RoboDK station: Sheet C - Top.rdk

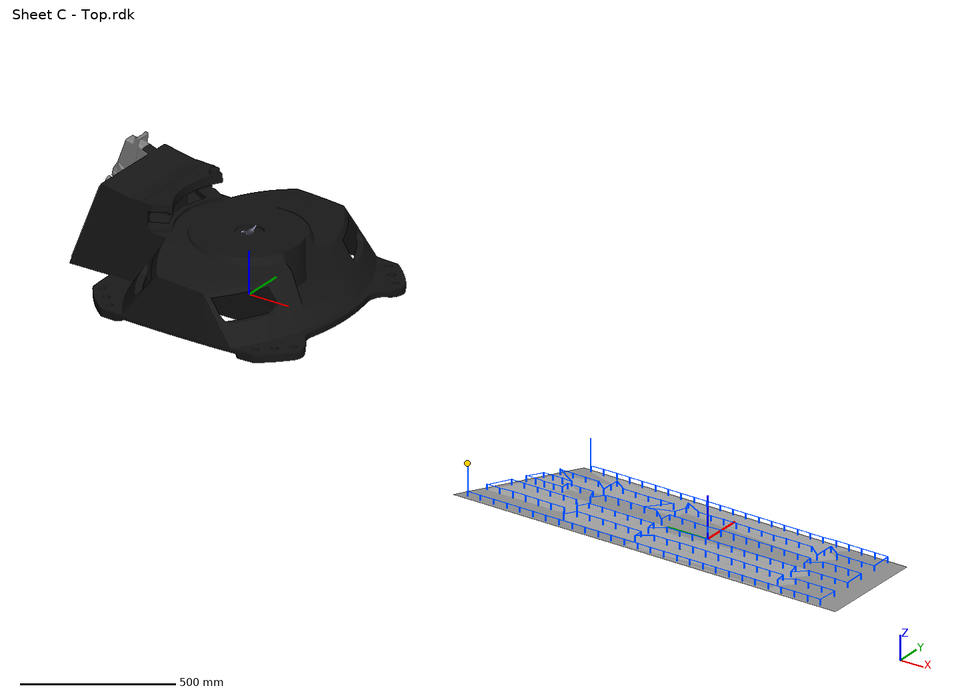
[picture v0: the station drawn from its stored meshes, robots at their saved joint values, targets as dots, program paths as lines]
Station Sheet C - Top (saved by RoboDK 5.2.3). Poses are relative to the parent item; angles as X-Y-Z fixed-axis rotations.
  - frame KUKA KR 210 R2700 extra Base at (0, 0, 0) mm
    - robot KUKA KR 210 R2700 extra: 6 axes, payload 210 kg, reach 2696 mm, repeatability 0.06 mm, weight 1068 kg
        joint limits [-185, -140, -120, -350, -125, -350] to [185, -5, 155, 350, 125, 350]; home [0, -90, 90, 0, 0, 0]; saved at [-11.417, -31.583, 137.817, -188.748, 54.991, -183.874]
      - tool Spindle, TCP at (32, 0, 260) mm, rotated rx 0 ry 39 rz 0 deg, size 157.3 x 72 x 259.9 mm
  - frame Frame 2 at (1800, 0, -372.68) mm, rotated rx 0 ry 0 rz 90 deg
    - object Box 1 - Sheet C -  Top at (0, 0, 0) mm, size 400 x 1500 x 0.8 mm, 1 curves, geometry from Box 1 - Sheet C -  Top.stl
    - object Sheet C-box 1 Hole positioning Top at (0, 0, 0) mm, 181 curves, geometry from Point 181
  - machining project Point settings: rotZ(0) | rotX(0)*rotY(0) | rotz(0)
  - program Point (916 instructions, listed below)
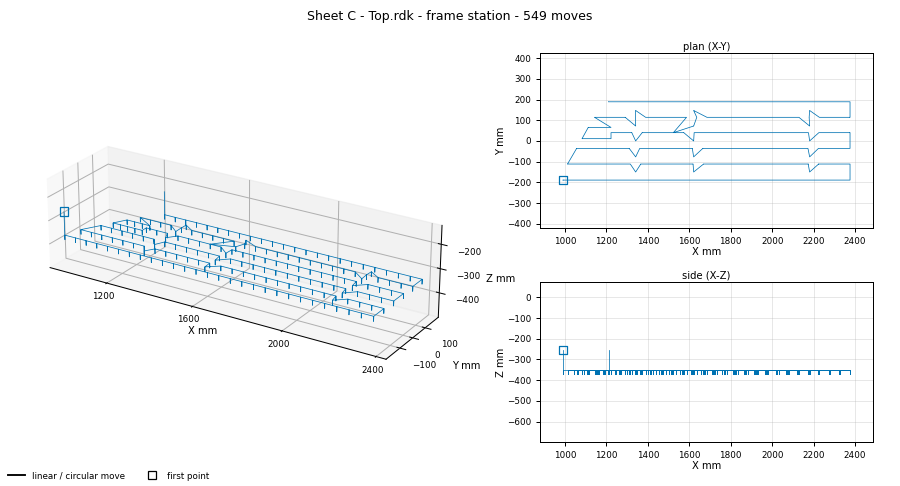
[picture p0: tool path of Sheet C - Top.rdk in frame station, 549 of 549 moves have a stored position in this frame; points joined in program order, loops and branches not executed]

--- program Point (robot KUKA KR 210 R2700 extra) ---
  Smooth(1)
  Set speed (1000.0 mm/s)
  Set Ref.: Frame 2
  Set Tool: Spindle
  Show Spindle
  MoveJ 1 to (-189, 810.01, 120) mm, rotated rx -180 ry 0 rz 90 deg; joints [14.788, -23.755, 145.264, -170.148, 69.845, -171.831]
  MoveL 2 to (-189, 810.01, 120) mm, rotated rx -180 ry 0 rz 90 deg; joints [14.788, -23.755, 145.264, -170.148, 69.845, -171.831]
  MoveL 3 to (-189, 810.01, 20) mm, rotated rx 180 ry 0 rz 90 deg; joints [14.788, -16.611, 140.997, -170.313, 72.681, -171.315]
  MoveL 4 to (-189, 810.01, 20) mm, rotated rx 180 ry 0 rz 90 deg; joints [14.788, -16.611, 140.997, -170.313, 72.681, -171.315]
  Set speed (50.0 mm/s)
  MoveL 5 to (-189, 810.01, 0) mm, rotated rx 180 ry 0 rz 90 deg; joints [14.788, -15.296, 140.112, -170.336, 73.105, -171.239]
  MoveL 6 to (-189, 810.01, 20) mm, rotated rx 180 ry 0 rz 90 deg; joints [14.788, -16.611, 140.997, -170.313, 72.681, -171.315]
  Set speed (1000.0 mm/s)
  MoveL 7 to (-189, 758.68, 20) mm, rotated rx 180 ry 0 rz 90 deg; joints [13.838, -18.904, 139.596, -170.729, 69.122, -172.492]
  Set speed (50.0 mm/s)
  MoveL 8 to (-189, 758.68, 0) mm, rotated rx -180 ry 0 rz 90 deg; joints [13.838, -17.57, 138.739, -170.758, 69.592, -172.41]
  MoveL 9 to (-189, 758.68, 20) mm, rotated rx 180 ry 0 rz 90 deg; joints [13.838, -18.904, 139.596, -170.729, 69.122, -172.492]
  Set speed (1000.0 mm/s)
  MoveL 10 to (-189, 707.34, 20) mm, rotated rx -180 ry 0 rz 90 deg; joints [13.001, -20.924, 138.071, -171.063, 65.686, -173.533]
  Set speed (50.0 mm/s)
  MoveL 11 to (-189, 707.34, 0) mm, rotated rx 180 ry 0 rz 90 deg; joints [13.001, -19.583, 137.241, -171.098, 66.19, -173.446]
  MoveL 12 to (-189, 707.34, 20) mm, rotated rx -180 ry 0 rz 90 deg; joints [13.001, -20.924, 138.071, -171.063, 65.686, -173.533]
  Set speed (1000.0 mm/s)
  MoveL 13 to (-189, 656.01, 20) mm, rotated rx 180 ry 0 rz 90 deg; joints [12.258, -22.682, 136.432, -171.327, 62.377, -174.462]
  Set speed (50.0 mm/s)
  MoveL 14 to (-189, 656.01, 0) mm, rotated rx 180 ry 0 rz 90 deg; joints [12.258, -21.344, 135.628, -171.369, 62.906, -174.371]
  MoveL 15 to (-189, 656.01, 20) mm, rotated rx 180 ry 0 rz 90 deg; joints [12.258, -22.682, 136.432, -171.327, 62.377, -174.462]
  Set speed (1000.0 mm/s)
  MoveL 16 to (-189, 604.68, 20) mm, rotated rx -180 ry 0 rz 90 deg; joints [11.594, -24.194, 134.688, -171.533, 59.195, -175.301]
  Set speed (50.0 mm/s)
  MoveL 17 to (-189, 604.68, 0) mm, rotated rx -180 ry 0 rz 90 deg; joints [11.594, -22.864, 133.91, -171.58, 59.74, -175.207]
  MoveL 18 to (-189, 604.68, 20) mm, rotated rx -180 ry 0 rz 90 deg; joints [11.594, -24.194, 134.688, -171.533, 59.195, -175.301]
  Set speed (1000.0 mm/s)
  MoveL 19 to (-189, 553.34, 20) mm, rotated rx -180 ry 0 rz 90 deg; joints [10.997, -25.475, 132.846, -171.687, 56.133, -176.067]
  Set speed (50.0 mm/s)
  MoveL 20 to (-189, 553.34, 0) mm, rotated rx 180 ry 0 rz 90 deg; joints [10.997, -24.16, 132.092, -171.741, 56.688, -175.97]
  MoveL 21 to (-189, 553.34, 20) mm, rotated rx -180 ry 0 rz 90 deg; joints [10.997, -25.475, 132.846, -171.687, 56.133, -176.067]
  Set speed (1000.0 mm/s)
  MoveL 22 to (-189, 502.01, 20) mm, rotated rx 180 ry 0 rz 90 deg; joints [10.458, -26.541, 130.913, -171.797, 53.186, -176.774]
  Set speed (50.0 mm/s)
  MoveL 23 to (-189, 502.01, 0) mm, rotated rx 180 ry 0 rz 90 deg; joints [10.458, -25.246, 130.183, -171.856, 53.746, -176.674]
  MoveL 24 to (-189, 502.01, 20) mm, rotated rx 180 ry 0 rz 90 deg; joints [10.458, -26.541, 130.913, -171.797, 53.186, -176.774]
  Set speed (1000.0 mm/s)
  MoveL 25 to (-189, 450.68, 20) mm, rotated rx -180 ry 0 rz 90 deg; joints [9.969, -27.41, 128.897, -171.865, 50.346, -177.434]
  Set speed (50.0 mm/s)
  MoveL 26 to (-189, 450.68, 0) mm, rotated rx 180 ry 0 rz 90 deg; joints [9.969, -26.137, 128.189, -171.931, 50.906, -177.33]
  MoveL 27 to (-189, 450.68, 20) mm, rotated rx -180 ry 0 rz 90 deg; joints [9.969, -27.41, 128.897, -171.865, 50.346, -177.434]
  Set speed (1000.0 mm/s)
  MoveL 28 to (-189, 399.34, 20) mm, rotated rx -180 ry 0 rz 90 deg; joints [9.523, -28.095, 126.8, -171.895, 47.604, -178.057]
  Set speed (50.0 mm/s)
  MoveL 29 to (-189, 399.34, 0) mm, rotated rx 180 ry 0 rz 90 deg; joints [9.523, -26.846, 126.113, -171.966, 48.16, -177.951]
  MoveL 30 to (-189, 399.34, 20) mm, rotated rx -180 ry 0 rz 90 deg; joints [9.523, -28.095, 126.8, -171.895, 47.604, -178.057]
  Set speed (1000.0 mm/s)
  MoveL 31 to (-189, 348.01, 20) mm, rotated rx 180 ry 0 rz 90 deg; joints [9.115, -28.611, 124.629, -171.887, 44.95, -178.653]
  Set speed (50.0 mm/s)
  MoveL 32 to (-189, 348.01, 0) mm, rotated rx 180 ry 0 rz 90 deg; joints [9.115, -27.388, 123.961, -171.965, 45.5, -178.543]
  MoveL 33 to (-189, 348.01, 20) mm, rotated rx 180 ry 0 rz 90 deg; joints [9.115, -28.611, 124.629, -171.887, 44.95, -178.653]
  Set speed (1000.0 mm/s)
  MoveL 34 to (-189, 296.68, 20) mm, rotated rx 180 ry 0 rz 90 deg; joints [8.741, -28.971, 122.385, -171.843, 42.377, -179.231]
  Set speed (50.0 mm/s)
  MoveL 35 to (-189, 296.68, 0) mm, rotated rx 180 ry 0 rz 90 deg; joints [8.741, -27.775, 121.736, -171.927, 42.919, -179.117]
  MoveL 36 to (-189, 296.68, 20) mm, rotated rx 180 ry 0 rz 90 deg; joints [8.741, -28.971, 122.385, -171.843, 42.377, -179.231]
  Set speed (1000.0 mm/s)
  MoveL 37 to (-189, 245.34, 20) mm, rotated rx 180 ry 0 rz 90 deg; joints [8.395, -29.188, 120.072, -171.76, 39.875, -179.799]
  Set speed (50.0 mm/s)
  MoveL 38 to (-189, 245.34, 0) mm, rotated rx 180 ry 0 rz 90 deg; joints [8.395, -28.018, 119.439, -171.851, 40.406, -179.68]
  MoveL 39 to (-189, 245.34, 20) mm, rotated rx 180 ry 0 rz 90 deg; joints [8.395, -29.188, 120.072, -171.76, 39.875, -179.799]
  Set speed (1000.0 mm/s)
  MoveL 40 to (-189, 194.01, 20) mm, rotated rx -180 ry 0 rz 90 deg; joints [8.076, -29.271, 117.69, -171.637, 37.436, -180.365]
  Set speed (50.0 mm/s)
  MoveL 41 to (-189, 194.01, 0) mm, rotated rx -180 ry 0 rz 90 deg; joints [8.076, -28.128, 117.073, -171.735, 37.956, -180.241]
  MoveL 42 to (-189, 194.01, 20) mm, rotated rx -180 ry 0 rz 90 deg; joints [8.076, -29.271, 117.69, -171.637, 37.436, -180.365]
  Set speed (1000.0 mm/s)
  MoveL 43 to (-189, 142.68, 20) mm, rotated rx -180 ry 0 rz 90 deg; joints [7.78, -29.229, 115.242, -171.469, 35.053, -180.939]
  Set speed (50.0 mm/s)
  MoveL 44 to (-189, 142.68, 0) mm, rotated rx 180 ry 0 rz 90 deg; joints [7.78, -28.112, 114.639, -171.576, 35.561, -180.808]
  MoveL 45 to (-189, 142.68, 20) mm, rotated rx -180 ry 0 rz 90 deg; joints [7.78, -29.229, 115.242, -171.469, 35.053, -180.939]
  Set speed (1000.0 mm/s)
  MoveL 46 to (-189, 91.34, 20) mm, rotated rx -180 ry 0 rz 90 deg; joints [7.505, -29.071, 112.726, -171.253, 32.718, -181.53]
  Set speed (50.0 mm/s)
  MoveL 47 to (-189, 91.34, 0) mm, rotated rx 180 ry 0 rz 90 deg; joints [7.505, -27.98, 112.135, -171.369, 33.212, -181.392]
  MoveL 48 to (-189, 91.34, 20) mm, rotated rx -180 ry 0 rz 90 deg; joints [7.505, -29.071, 112.726, -171.253, 32.718, -181.53]
  Set speed (1000.0 mm/s)
  MoveL 49 to (-189, 40.01, 20) mm, rotated rx -180 ry 0 rz 90 deg; joints [7.249, -28.804, 110.142, -170.978, 30.424, -182.151]
  Set speed (50.0 mm/s)
  MoveL 50 to (-189, 40.01, 0) mm, rotated rx -180 ry 0 rz 90 deg; joints [7.249, -27.738, 109.563, -171.106, 30.905, -182.002]
  MoveL 51 to (-189, 40.01, 20) mm, rotated rx -180 ry 0 rz 90 deg; joints [7.249, -28.804, 110.142, -170.978, 30.424, -182.151]
  Set speed (1000.0 mm/s)
  MoveL 52 to (-189, -11.32, 20) mm, rotated rx 180 ry 0 rz 90 deg; joints [7.009, -28.434, 107.49, -170.637, 28.165, -182.813]
  Set speed (50.0 mm/s)
  MoveL 53 to (-189, -11.32, 0) mm, rotated rx -180 ry 0 rz 90 deg; joints [7.009, -27.391, 106.92, -170.778, 28.632, -182.653]
  MoveL 54 to (-189, -11.32, 20) mm, rotated rx 180 ry 0 rz 90 deg; joints [7.009, -28.434, 107.49, -170.637, 28.165, -182.813]
  Set speed (1000.0 mm/s)
  MoveL 55 to (-189, -62.66, 20) mm, rotated rx 180 ry 0 rz 90 deg; joints [6.785, -27.964, 104.766, -170.212, 25.933, -183.536]
  Set speed (50.0 mm/s)
  MoveL 56 to (-189, -62.66, 0) mm, rotated rx 180 ry 0 rz 90 deg; joints [6.785, -26.945, 104.205, -170.369, 26.385, -183.361]
  MoveL 57 to (-189, -62.66, 20) mm, rotated rx 180 ry 0 rz 90 deg; joints [6.785, -27.964, 104.766, -170.212, 25.933, -183.536]
  Set speed (1000.0 mm/s)
  MoveL 58 to (-189, -113.99, 20) mm, rotated rx 180 ry 0 rz 90 deg; joints [6.574, -27.401, 101.968, -169.684, 23.725, -184.343]
  Set speed (50.0 mm/s)
  MoveL 59 to (-189, -113.99, 0) mm, rotated rx -180 ry 0 rz 90 deg; joints [6.574, -26.403, 101.414, -169.861, 24.162, -184.148]
  MoveL 60 to (-189, -113.99, 20) mm, rotated rx 180 ry 0 rz 90 deg; joints [6.574, -27.401, 101.968, -169.684, 23.725, -184.343]
  Set speed (1000.0 mm/s)
  MoveL 61 to (-189, -165.32, 20) mm, rotated rx -180 ry 0 rz 90 deg; joints [6.376, -26.745, 99.093, -169.022, 21.533, -185.265]
  Set speed (50.0 mm/s)
  MoveL 62 to (-189, -165.32, 0) mm, rotated rx -180 ry 0 rz 90 deg; joints [6.376, -25.768, 98.545, -169.226, 21.955, -185.046]
  MoveL 63 to (-189, -165.32, 20) mm, rotated rx -180 ry 0 rz 90 deg; joints [6.376, -26.745, 99.093, -169.022, 21.533, -185.265]
  Set speed (1000.0 mm/s)
  MoveL 64 to (-189, -216.66, 20) mm, rotated rx 180 ry 0 rz 90 deg; joints [6.19, -26, 96.135, -168.183, 19.352, -186.348]
  Set speed (50.0 mm/s)
  MoveL 65 to (-189, -216.66, 0) mm, rotated rx -180 ry 0 rz 90 deg; joints [6.19, -25.042, 95.592, -168.42, 19.758, -186.097]
  MoveL 66 to (-189, -216.66, 20) mm, rotated rx 180 ry 0 rz 90 deg; joints [6.19, -26, 96.135, -168.183, 19.352, -186.348]
  Set speed (1000.0 mm/s)
  MoveL 67 to (-189, -267.99, 20) mm, rotated rx 180 ry 0 rz 90 deg; joints [6.014, -25.166, 93.09, -167.099, 17.178, -187.662]
  Set speed (50.0 mm/s)
  MoveL 68 to (-189, -267.99, 0) mm, rotated rx 180 ry 0 rz 90 deg; joints [6.014, -24.226, 92.55, -167.382, 17.568, -187.366]
  MoveL 69 to (-189, -267.99, 20) mm, rotated rx 180 ry 0 rz 90 deg; joints [6.014, -25.166, 93.09, -167.099, 17.178, -187.662]
  Set speed (1000.0 mm/s)
  MoveL 70 to (-189, -319.32, 20) mm, rotated rx -180 ry 0 rz 90 deg; joints [5.848, -24.243, 89.949, -165.662, 15.007, -189.317]
  Set speed (50.0 mm/s)
  MoveL 71 to (-189, -319.32, 0) mm, rotated rx -180 ry 0 rz 90 deg; joints [5.848, -23.32, 89.411, -166.009, 15.38, -188.957]
  MoveL 72 to (-189, -319.32, 20) mm, rotated rx -180 ry 0 rz 90 deg; joints [5.848, -24.243, 89.949, -165.662, 15.007, -189.317]
  Set speed (1000.0 mm/s)
  MoveL 73 to (-189, -370.66, 20) mm, rotated rx 180 ry 0 rz 90 deg; joints [5.691, -23.23, 86.705, -163.687, 12.837, -191.497]
  Set speed (50.0 mm/s)
  MoveL 74 to (-189, -370.66, 0) mm, rotated rx 180 ry 0 rz 90 deg; joints [5.691, -22.323, 86.167, -164.131, 13.192, -191.043]
  MoveL 75 to (-189, -370.66, 20) mm, rotated rx 180 ry 0 rz 90 deg; joints [5.691, -23.23, 86.705, -163.687, 12.837, -191.497]
  Set speed (1000.0 mm/s)
  MoveL 76 to (-189, -421.99, 20) mm, rotated rx -180 ry 0 rz 90 deg; joints [5.542, -22.125, 83.347, -160.837, 10.67, -194.543]
  Set speed (50.0 mm/s)
  MoveL 77 to (-189, -421.99, 0) mm, rotated rx 180 ry 0 rz 90 deg; joints [5.542, -21.231, 82.807, -161.435, 11.004, -193.935]
  MoveL 78 to (-189, -421.99, 20) mm, rotated rx -180 ry 0 rz 90 deg; joints [5.542, -22.125, 83.347, -160.837, 10.67, -194.543]
  Set speed (1000.0 mm/s)
  MoveL 79 to (-189, -473.32, 20) mm, rotated rx 180 ry 0 rz 90 deg; joints [5.4, -20.924, 79.863, -156.425, 8.516, -199.141]
  Set speed (50.0 mm/s)
  MoveL 80 to (-189, -473.32, 0) mm, rotated rx -180 ry 0 rz 90 deg; joints [5.4, -20.042, 79.319, -157.295, 8.827, -198.261]
  MoveL 81 to (-189, -473.32, 20) mm, rotated rx 180 ry 0 rz 90 deg; joints [5.4, -20.924, 79.863, -156.425, 8.516, -199.141]
  Set speed (1000.0 mm/s)
  MoveL 82 to (-189, -524.66, 20) mm, rotated rx -180 ry 0 rz 90 deg; joints [5.266, -19.621, 76.236, -148.871, 6.415, -206.873]
  Set speed (50.0 mm/s)
  MoveL 83 to (-189, -524.66, 0) mm, rotated rx -180 ry 0 rz 90 deg; joints [5.266, -18.75, 75.686, -150.285, 6.691, -205.45]
  MoveL 84 to (-189, -524.66, 20) mm, rotated rx -180 ry 0 rz 90 deg; joints [5.266, -19.621, 76.236, -148.871, 6.415, -206.873]
  Set speed (1000.0 mm/s)
  MoveL 85 to (-189, -575.99, 20) mm, rotated rx -180 ry 0 rz 90 deg; joints [5.138, -18.208, 72.448, -134.025, 4.496, -221.889]
  Set speed (50.0 mm/s)
  MoveL 86 to (-189, -575.99, 0) mm, rotated rx 180 ry 0 rz 90 deg; joints [5.138, -17.345, 71.889, -136.67, 4.711, -219.236]
  MoveL 87 to (-189, -575.99, 20) mm, rotated rx -180 ry 0 rz 90 deg; joints [5.138, -18.208, 72.448, -134.025, 4.496, -221.889]
  Set speed (1000.0 mm/s)
  MoveL 88 to (-111.5, -575.99, 20) mm, rotated rx 180 ry 0 rz 90 deg; joints [3.036, -18.366, 72.866, -151.076, 3.952, -206.505]
  Set speed (50.0 mm/s)
  MoveL 89 to (-111.5, -575.99, 0) mm, rotated rx -180 ry 0 rz 90 deg; joints [3.036, -17.503, 72.308, -153.075, 4.222, -204.502]
  MoveL 90 to (-111.5, -575.99, 20) mm, rotated rx 180 ry 0 rz 90 deg; joints [3.036, -18.366, 72.866, -151.076, 3.952, -206.505]
  Set speed (1000.0 mm/s)
  MoveL 91 to (-111.5, -525.47, 20) mm, rotated rx 180 ry 0 rz 90 deg; joints [3.111, -19.749, 76.587, -161.307, 6.118, -196.175]
  Set speed (50.0 mm/s)
  MoveL 92 to (-111.5, -525.47, 0) mm, rotated rx 180 ry 0 rz 90 deg; joints [3.111, -18.877, 76.038, -162.225, 6.424, -195.252]
  MoveL 93 to (-111.5, -525.47, 20) mm, rotated rx 180 ry 0 rz 90 deg; joints [3.111, -19.749, 76.587, -161.307, 6.118, -196.175]
  Set speed (1000.0 mm/s)
  MoveL 94 to (-111.5, -474.95, 20) mm, rotated rx 180 ry 0 rz 90 deg; joints [3.19, -21.026, 80.154, -166.01, 8.328, -191.369]
  Set speed (50.0 mm/s)
  MoveL 95 to (-111.5, -474.95, 0) mm, rotated rx 180 ry 0 rz 90 deg; joints [3.19, -20.144, 79.61, -166.548, 8.657, -190.824]
  MoveL 96 to (-111.5, -474.95, 20) mm, rotated rx 180 ry 0 rz 90 deg; joints [3.19, -21.026, 80.154, -166.01, 8.328, -191.369]
  Set speed (1000.0 mm/s)
  MoveL 97 to (-111.5, -424.43, 20) mm, rotated rx -180 ry 0 rz 90 deg; joints [3.272, -22.205, 83.583, -168.669, 10.533, -188.601]
  Set speed (50.0 mm/s)
  MoveL 98 to (-111.5, -424.43, 0) mm, rotated rx -180 ry 0 rz 90 deg; joints [3.272, -21.31, 83.043, -169.032, 10.882, -188.232]
  MoveL 99 to (-111.5, -424.43, 20) mm, rotated rx -180 ry 0 rz 90 deg; joints [3.272, -22.205, 83.583, -168.669, 10.533, -188.601]
  Set speed (1000.0 mm/s)
  MoveL 100 to (-150, -380.99, 20) mm, rotated rx 180 ry 0 rz 90 deg; joints [4.498, -23.088, 86.263, -166.725, 12.41, -189.478]
  Set speed (50.0 mm/s)
  MoveL 101 to (-150, -380.99, 0) mm, rotated rx -180 ry 0 rz 90 deg; joints [4.498, -22.182, 85.725, -167.097, 12.768, -189.096]
  MoveL 102 to (-150, -380.99, 20) mm, rotated rx 180 ry 0 rz 90 deg; joints [4.498, -23.088, 86.263, -166.725, 12.41, -189.478]
  Set speed (1000.0 mm/s)
  MoveL 103 to (-111.5, -373.92, 20) mm, rotated rx -180 ry 0 rz 90 deg; joints [3.359, -23.29, 86.89, -170.365, 12.726, -186.791]
  Set speed (50.0 mm/s)
  MoveL 104 to (-111.5, -373.92, 0) mm, rotated rx 180 ry 0 rz 90 deg; joints [3.359, -22.381, 86.352, -170.632, 13.091, -186.518]
  MoveL 105 to (-111.5, -373.92, 20) mm, rotated rx -180 ry 0 rz 90 deg; joints [3.359, -23.29, 86.89, -170.365, 12.726, -186.791]
  Set speed (1000.0 mm/s)
  MoveL 106 to (-111.5, -323.4, 20) mm, rotated rx 180 ry 0 rz 90 deg; joints [3.45, -24.285, 90.088, -171.534, 14.907, -185.503]
  Set speed (50.0 mm/s)
  MoveL 107 to (-111.5, -323.4, 0) mm, rotated rx 180 ry 0 rz 90 deg; joints [3.45, -23.361, 89.549, -171.742, 15.288, -185.287]
  MoveL 108 to (-111.5, -323.4, 20) mm, rotated rx 180 ry 0 rz 90 deg; joints [3.45, -24.285, 90.088, -171.534, 14.907, -185.503]
  Set speed (1000.0 mm/s)
  MoveL 109 to (-111.5, -272.88, 20) mm, rotated rx 180 ry 0 rz 90 deg; joints [3.547, -25.193, 93.186, -172.383, 17.081, -184.527]
  Set speed (50.0 mm/s)
  MoveL 110 to (-111.5, -272.88, 0) mm, rotated rx 180 ry 0 rz 90 deg; joints [3.547, -24.253, 92.646, -172.552, 17.478, -184.35]
  MoveL 111 to (-111.5, -272.88, 20) mm, rotated rx 180 ry 0 rz 90 deg; joints [3.547, -25.193, 93.186, -172.383, 17.081, -184.527]
  Set speed (1000.0 mm/s)
  MoveL 112 to (-111.5, -222.36, 20) mm, rotated rx 180 ry 0 rz 90 deg; joints [3.649, -26.015, 96.192, -173.023, 19.252, -183.753]
  Set speed (50.0 mm/s)
  MoveL 113 to (-111.5, -222.36, 0) mm, rotated rx -180 ry 0 rz 90 deg; joints [3.649, -25.056, 95.649, -173.164, 19.664, -183.603]
  MoveL 114 to (-111.5, -222.36, 20) mm, rotated rx 180 ry 0 rz 90 deg; joints [3.649, -26.015, 96.192, -173.023, 19.252, -183.753]
  Set speed (1000.0 mm/s)
  MoveL 115 to (-111.5, -171.84, 20) mm, rotated rx 180 ry 0 rz 90 deg; joints [3.757, -26.75, 99.113, -173.518, 21.427, -183.116]
  Set speed (50.0 mm/s)
  MoveL 116 to (-111.5, -171.84, 0) mm, rotated rx 180 ry 0 rz 90 deg; joints [3.757, -25.772, 98.565, -173.639, 21.854, -182.985]
  MoveL 117 to (-111.5, -171.84, 20) mm, rotated rx 180 ry 0 rz 90 deg; joints [3.757, -26.75, 99.113, -173.518, 21.427, -183.116]
  Set speed (1000.0 mm/s)
  MoveL 118 to (-111.5, -121.32, 20) mm, rotated rx -180 ry 0 rz 90 deg; joints [3.872, -27.398, 101.954, -173.909, 23.611, -182.573]
  Set speed (50.0 mm/s)
  MoveL 119 to (-111.5, -121.32, 0) mm, rotated rx -180 ry 0 rz 90 deg; joints [3.872, -26.4, 101.401, -174.015, 24.053, -182.458]
  MoveL 120 to (-111.5, -121.32, 20) mm, rotated rx -180 ry 0 rz 90 deg; joints [3.872, -27.398, 101.954, -173.909, 23.611, -182.573]
  Set speed (1000.0 mm/s)
  MoveL 121 to (-111.5, -70.81, 20) mm, rotated rx 180 ry 0 rz 90 deg; joints [3.994, -27.956, 104.72, -174.221, 25.811, -182.099]
  Set speed (50.0 mm/s)
  MoveL 122 to (-111.5, -70.81, 0) mm, rotated rx 180 ry 0 rz 90 deg; joints [3.994, -26.937, 104.16, -174.315, 26.267, -181.995]
  MoveL 123 to (-111.5, -70.81, 20) mm, rotated rx 180 ry 0 rz 90 deg; joints [3.994, -27.956, 104.72, -174.221, 25.811, -182.099]
  Set speed (1000.0 mm/s)
  MoveL 124 to (-111.5, -20.29, 20) mm, rotated rx 180 ry 0 rz 90 deg; joints [4.125, -28.422, 107.415, -174.473, 28.031, -181.674]
  Set speed (50.0 mm/s)
  MoveL 125 to (-111.5, -20.29, 0) mm, rotated rx -180 ry 0 rz 90 deg; joints [4.125, -27.38, 106.846, -174.557, 28.502, -181.579]
  MoveL 126 to (-111.5, -20.29, 20) mm, rotated rx 180 ry 0 rz 90 deg; joints [4.125, -28.422, 107.415, -174.473, 28.031, -181.674]
  Set speed (1000.0 mm/s)
  MoveL 127 to (-111.5, 30.23, 20) mm, rotated rx -180 ry 0 rz 90 deg; joints [4.263, -28.792, 110.042, -174.676, 30.28, -181.285]
  Set speed (50.0 mm/s)
  MoveL 128 to (-111.5, 30.23, 0) mm, rotated rx -180 ry 0 rz 90 deg; joints [4.263, -27.726, 109.462, -174.752, 30.764, -181.197]
  MoveL 129 to (-111.5, 30.23, 20) mm, rotated rx -180 ry 0 rz 90 deg; joints [4.263, -28.792, 110.042, -174.676, 30.28, -181.285]
  Set speed (1000.0 mm/s)
  MoveL 130 to (-111.5, 80.75, 20) mm, rotated rx -180 ry 0 rz 90 deg; joints [4.412, -29.061, 112.601, -174.84, 32.563, -180.921]
  Set speed (50.0 mm/s)
  MoveL 131 to (-111.5, 80.75, 0) mm, rotated rx 180 ry 0 rz 90 deg; joints [4.412, -27.971, 112.011, -174.909, 33.06, -180.839]
  MoveL 132 to (-111.5, 80.75, 20) mm, rotated rx -180 ry 0 rz 90 deg; joints [4.412, -29.061, 112.601, -174.84, 32.563, -180.921]
  Set speed (1000.0 mm/s)
  MoveL 133 to (-111.5, 131.27, 20) mm, rotated rx -180 ry 0 rz 90 deg; joints [4.571, -29.223, 115.095, -174.97, 34.887, -180.575]
  Set speed (50.0 mm/s)
  MoveL 134 to (-111.5, 131.27, 0) mm, rotated rx -180 ry 0 rz 90 deg; joints [4.571, -28.108, 114.492, -175.033, 35.397, -180.497]
  MoveL 135 to (-111.5, 131.27, 20) mm, rotated rx -180 ry 0 rz 90 deg; joints [4.571, -29.223, 115.095, -174.97, 34.887, -180.575]
  Set speed (1000.0 mm/s)
  MoveL 136 to (-150, 179.01, 20) mm, rotated rx -180 ry 0 rz 90 deg; joints [6.355, -29.272, 117.215, -173.347, 36.956, -180.379]
  Set speed (50.0 mm/s)
  MoveL 137 to (-150, 179.01, 0) mm, rotated rx 180 ry 0 rz 90 deg; joints [6.355, -28.134, 116.6, -173.426, 37.476, -180.279]
  MoveL 138 to (-150, 179.01, 20) mm, rotated rx -180 ry 0 rz 90 deg; joints [6.355, -29.272, 117.215, -173.347, 36.956, -180.379]
  Set speed (1000.0 mm/s)
  MoveL 139 to (-111.5, 181.79, 20) mm, rotated rx 180 ry 0 rz 90 deg; joints [4.742, -29.272, 117.524, -175.07, 37.259, -180.239]
  Set speed (50.0 mm/s)
  MoveL 140 to (-111.5, 181.79, 0) mm, rotated rx -180 ry 0 rz 90 deg; joints [4.742, -28.13, 116.908, -175.129, 37.782, -180.165]
  MoveL 141 to (-111.5, 181.79, 20) mm, rotated rx 180 ry 0 rz 90 deg; joints [4.742, -29.272, 117.524, -175.07, 37.259, -180.239]
  Set speed (1000.0 mm/s)
  MoveL 142 to (-111.5, 232.31, 20) mm, rotated rx -180 ry 0 rz 90 deg; joints [4.926, -29.199, 119.889, -175.145, 39.687, -179.907]
  Set speed (50.0 mm/s)
  MoveL 143 to (-111.5, 232.31, 0) mm, rotated rx 180 ry 0 rz 90 deg; joints [4.926, -28.031, 119.257, -175.199, 40.222, -179.837]
  MoveL 144 to (-111.5, 232.31, 20) mm, rotated rx -180 ry 0 rz 90 deg; joints [4.926, -29.199, 119.889, -175.145, 39.687, -179.907]
  Set speed (1000.0 mm/s)
  MoveL 145 to (-111.5, 282.82, 20) mm, rotated rx 180 ry 0 rz 90 deg; joints [5.125, -28.996, 122.187, -175.197, 42.179, -179.576]
  Set speed (50.0 mm/s)
  MoveL 146 to (-111.5, 282.82, 0) mm, rotated rx 180 ry 0 rz 90 deg; joints [5.125, -27.802, 121.539, -175.247, 42.724, -179.508]
  MoveL 147 to (-111.5, 282.82, 20) mm, rotated rx 180 ry 0 rz 90 deg; joints [5.125, -28.996, 122.187, -175.197, 42.179, -179.576]
  Set speed (1000.0 mm/s)
  MoveL 148 to (-111.5, 333.34, 20) mm, rotated rx -180 ry 0 rz 90 deg; joints [5.341, -28.652, 124.419, -175.226, 44.745, -179.239]
  Set speed (50.0 mm/s)
  MoveL 149 to (-111.5, 333.34, 0) mm, rotated rx 180 ry 0 rz 90 deg; joints [5.341, -27.431, 123.754, -175.272, 45.298, -179.174]
  MoveL 150 to (-111.5, 333.34, 20) mm, rotated rx -180 ry 0 rz 90 deg; joints [5.341, -28.652, 124.419, -175.226, 44.745, -179.239]
  Set speed (1000.0 mm/s)
  MoveL 151 to (-111.5, 383.86, 20) mm, rotated rx -180 ry 0 rz 90 deg; joints [5.576, -28.155, 126.582, -175.234, 47.393, -178.891]
  Set speed (50.0 mm/s)
  MoveL 152 to (-111.5, 383.86, 0) mm, rotated rx 180 ry 0 rz 90 deg; joints [5.576, -26.909, 125.897, -175.277, 47.952, -178.829]
  MoveL 153 to (-111.5, 383.86, 20) mm, rotated rx -180 ry 0 rz 90 deg; joints [5.576, -28.155, 126.582, -175.234, 47.393, -178.891]
  Set speed (1000.0 mm/s)
  MoveL 154 to (-111.5, 434.38, 20) mm, rotated rx -180 ry 0 rz 90 deg; joints [5.832, -27.493, 128.672, -175.221, 50.133, -178.529]
  Set speed (50.0 mm/s)
  MoveL 155 to (-111.5, 434.38, 0) mm, rotated rx 180 ry 0 rz 90 deg; joints [5.832, -26.222, 127.967, -175.259, 50.696, -178.468]
  MoveL 156 to (-111.5, 434.38, 20) mm, rotated rx -180 ry 0 rz 90 deg; joints [5.832, -27.493, 128.672, -175.221, 50.133, -178.529]
  Set speed (1000.0 mm/s)
  MoveL 157 to (-150, 459.01, 20) mm, rotated rx 180 ry 0 rz 90 deg; joints [8.003, -27.183, 129.476, -173.545, 51.198, -177.82]
  Set speed (50.0 mm/s)
  MoveL 158 to (-150, 459.01, 0) mm, rotated rx -180 ry 0 rz 90 deg; joints [8.003, -25.903, 128.762, -173.595, 51.76, -177.739]
  MoveL 159 to (-150, 459.01, 20) mm, rotated rx 180 ry 0 rz 90 deg; joints [8.003, -27.183, 129.476, -173.545, 51.198, -177.82]
  Set speed (1000.0 mm/s)
  MoveL 160 to (-111.5, 484.9, 20) mm, rotated rx 180 ry 0 rz 90 deg; joints [6.113, -26.65, 130.687, -175.185, 52.975, -178.146]
  Set speed (50.0 mm/s)
  MoveL 161 to (-111.5, 484.9, 0) mm, rotated rx 180 ry 0 rz 90 deg; joints [6.113, -25.357, 129.96, -175.22, 53.538, -178.087]
  MoveL 162 to (-111.5, 484.9, 20) mm, rotated rx 180 ry 0 rz 90 deg; joints [6.113, -26.65, 130.687, -175.185, 52.975, -178.146]
  Set speed (1000.0 mm/s)
  MoveL 163 to (-111.5, 535.42, 20) mm, rotated rx -180 ry 0 rz 90 deg; joints [6.423, -25.612, 132.621, -175.125, 55.929, -177.736]
  Set speed (50.0 mm/s)
  MoveL 164 to (-111.5, 535.42, 0) mm, rotated rx 180 ry 0 rz 90 deg; joints [6.423, -24.3, 131.87, -175.157, 56.488, -177.679]
  MoveL 165 to (-111.5, 535.42, 20) mm, rotated rx -180 ry 0 rz 90 deg; joints [6.423, -25.612, 132.621, -175.125, 55.929, -177.736]
  Set speed (1000.0 mm/s)
  MoveL 166 to (-111.5, 585.94, 20) mm, rotated rx -180 ry 0 rz 90 deg; joints [6.765, -24.362, 134.468, -175.039, 59.005, -177.293]
  Set speed (50.0 mm/s)
  MoveL 167 to (-111.5, 585.94, 0) mm, rotated rx 180 ry 0 rz 90 deg; joints [6.765, -23.034, 133.693, -175.067, 59.556, -177.237]
  MoveL 168 to (-111.5, 585.94, 20) mm, rotated rx -180 ry 0 rz 90 deg; joints [6.765, -24.362, 134.468, -175.039, 59.005, -177.293]
  Set speed (1000.0 mm/s)
  MoveL 169 to (-111.5, 636.45, 20) mm, rotated rx 180 ry 0 rz 90 deg; joints [7.145, -22.883, 136.221, -174.924, 62.213, -176.807]
  Set speed (50.0 mm/s)
  MoveL 170 to (-111.5, 636.45, 0) mm, rotated rx 180 ry 0 rz 90 deg; joints [7.145, -21.545, 135.421, -174.949, 62.748, -176.754]
  MoveL 171 to (-111.5, 636.45, 20) mm, rotated rx 180 ry 0 rz 90 deg; joints [7.145, -22.883, 136.221, -174.924, 62.213, -176.807]
  Set speed (1000.0 mm/s)
  MoveL 172 to (-111.5, 686.97, 20) mm, rotated rx 180 ry 0 rz 90 deg; joints [7.57, -21.156, 137.874, -174.775, 65.563, -176.27]
  Set speed (50.0 mm/s)
  MoveL 173 to (-111.5, 686.97, 0) mm, rotated rx 180 ry 0 rz 90 deg; joints [7.57, -19.815, 137.047, -174.796, 66.074, -176.219]
  MoveL 174 to (-111.5, 686.97, 20) mm, rotated rx 180 ry 0 rz 90 deg; joints [7.57, -21.156, 137.874, -174.775, 65.563, -176.27]
  Set speed (1000.0 mm/s)
  MoveL 175 to (-111.5, 737.49, 20) mm, rotated rx -180 ry 0 rz 90 deg; joints [8.049, -19.165, 139.416, -174.586, 69.06, -175.668]
  Set speed (50.0 mm/s)
  MoveL 176 to (-111.5, 737.49, 0) mm, rotated rx -180 ry 0 rz 90 deg; joints [8.049, -17.831, 138.562, -174.603, 69.538, -175.62]
  MoveL 177 to (-111.5, 737.49, 20) mm, rotated rx -180 ry 0 rz 90 deg; joints [8.049, -19.165, 139.416, -174.586, 69.06, -175.668]
  Set speed (1000.0 mm/s)
  MoveL 178 to (-111.5, 788.01, 20) mm, rotated rx 180 ry 0 rz 90 deg; joints [8.592, -16.895, 140.838, -174.349, 72.706, -174.988]
  Set speed (50.0 mm/s)
  MoveL 179 to (-111.5, 788.01, 0) mm, rotated rx 180 ry 0 rz 90 deg; joints [8.592, -15.578, 139.957, -174.362, 73.141, -174.943]
  MoveL 180 to (-111.5, 788.01, 20) mm, rotated rx 180 ry 0 rz 90 deg; joints [8.592, -16.895, 140.838, -174.349, 72.706, -174.988]
  Set speed (1000.0 mm/s)
  MoveL 181 to (-36, 744.01, 20) mm, rotated rx -180 ry 0 rz 90 deg; joints [2.636, -18.579, 139.814, -178.237, 70.214, -178.548]
  Set speed (50.0 mm/s)
  MoveL 182 to (-36, 744.01, 0) mm, rotated rx 180 ry 0 rz 90 deg; joints [2.636, -17.248, 138.952, -178.242, 70.683, -178.532]
  MoveL 183 to (-36, 744.01, 20) mm, rotated rx -180 ry 0 rz 90 deg; joints [2.636, -18.579, 139.814, -178.237, 70.214, -178.548]
  Set speed (1000.0 mm/s)
  MoveL 184 to (-36, 693.24, 20) mm, rotated rx 180 ry 0 rz 90 deg; joints [2.476, -20.67, 138.281, -178.303, 66.594, -178.75]
  Set speed (50.0 mm/s)
  MoveL 185 to (-36, 693.24, 0) mm, rotated rx -180 ry 0 rz 90 deg; joints [2.476, -19.33, 137.447, -178.309, 67.1, -178.734]
  MoveL 186 to (-36, 693.24, 20) mm, rotated rx 180 ry 0 rz 90 deg; joints [2.476, -20.67, 138.281, -178.303, 66.594, -178.75]
  Set speed (1000.0 mm/s)
  MoveL 187 to (-36, 642.47, 20) mm, rotated rx 180 ry 0 rz 90 deg; joints [2.333, -22.484, 136.635, -178.354, 63.137, -178.93]
  Set speed (50.0 mm/s)
  MoveL 188 to (-36, 642.47, 0) mm, rotated rx -180 ry 0 rz 90 deg; joints [2.333, -21.145, 135.828, -178.362, 63.669, -178.913]
  MoveL 189 to (-36, 642.47, 20) mm, rotated rx 180 ry 0 rz 90 deg; joints [2.333, -22.484, 136.635, -178.354, 63.137, -178.93]
  Set speed (1000.0 mm/s)
  MoveL 190 to (-36, 591.7, 20) mm, rotated rx -180 ry 0 rz 90 deg; joints [2.207, -24.039, 134.884, -178.394, 59.834, -179.092]
  Set speed (50.0 mm/s)
  MoveL 191 to (-36, 591.7, 0) mm, rotated rx 180 ry 0 rz 90 deg; joints [2.207, -22.709, 134.103, -178.403, 60.383, -179.074]
  MoveL 192 to (-36, 591.7, 20) mm, rotated rx -180 ry 0 rz 90 deg; joints [2.207, -24.039, 134.884, -178.394, 59.834, -179.092]
  Set speed (1000.0 mm/s)
  MoveL 193 to (-36, 540.93, 20) mm, rotated rx -180 ry 0 rz 90 deg; joints [2.093, -25.355, 133.037, -178.424, 56.674, -179.239]
  Set speed (50.0 mm/s)
  MoveL 194 to (-36, 540.93, 0) mm, rotated rx -180 ry 0 rz 90 deg; joints [2.093, -24.038, 132.281, -178.434, 57.234, -179.221]
  MoveL 195 to (-36, 540.93, 20) mm, rotated rx -180 ry 0 rz 90 deg; joints [2.093, -25.355, 133.037, -178.424, 56.674, -179.239]
  Set speed (1000.0 mm/s)
  MoveL 196 to (-36, 490.16, 20) mm, rotated rx 180 ry 0 rz 90 deg; joints [1.991, -26.448, 131.102, -178.445, 53.646, -179.375]
  Set speed (50.0 mm/s)
  MoveL 197 to (-36, 490.16, 0) mm, rotated rx 180 ry 0 rz 90 deg; joints [1.991, -25.151, 130.37, -178.456, 54.211, -179.356]
  MoveL 198 to (-36, 490.16, 20) mm, rotated rx 180 ry 0 rz 90 deg; joints [1.991, -26.448, 131.102, -178.445, 53.646, -179.375]
  Set speed (1000.0 mm/s)
  MoveL 199 to (-77, 459.01, 20) mm, rotated rx -180 ry 0 rz 90 deg; joints [4.128, -27.054, 129.786, -176.691, 51.705, -178.842]
  Set speed (50.0 mm/s)
  MoveL 200 to (-77, 459.01, 0) mm, rotated rx -180 ry 0 rz 90 deg; joints [4.128, -25.771, 129.069, -176.717, 52.27, -178.801]
  MoveL 201 to (-77, 459.01, 20) mm, rotated rx -180 ry 0 rz 90 deg; joints [4.128, -27.054, 129.786, -176.691, 51.705, -178.842]
  Set speed (1000.0 mm/s)
  MoveL 202 to (-36, 439.39, 20) mm, rotated rx -180 ry 0 rz 90 deg; joints [1.898, -27.338, 129.083, -178.458, 50.74, -179.501]
  Set speed (50.0 mm/s)
  MoveL 203 to (-36, 439.39, 0) mm, rotated rx 180 ry 0 rz 90 deg; joints [1.898, -26.063, 128.374, -178.47, 51.305, -179.482]
  MoveL 204 to (-36, 439.39, 20) mm, rotated rx -180 ry 0 rz 90 deg; joints [1.898, -27.338, 129.083, -178.458, 50.74, -179.501]
  Set speed (1000.0 mm/s)
  MoveL 205 to (-36, 388.63, 20) mm, rotated rx 180 ry 0 rz 90 deg; joints [1.813, -28.041, 126.988, -178.463, 47.943, -179.62]
  Set speed (50.0 mm/s)
  MoveL 206 to (-36, 388.63, 0) mm, rotated rx -180 ry 0 rz 90 deg; joints [1.813, -26.791, 126.299, -178.477, 48.505, -179.6]
  MoveL 207 to (-36, 388.63, 20) mm, rotated rx 180 ry 0 rz 90 deg; joints [1.813, -28.041, 126.988, -178.463, 47.943, -179.62]
  Set speed (1000.0 mm/s)
  MoveL 208 to (-36, 337.86, 20) mm, rotated rx 180 ry 0 rz 90 deg; joints [1.736, -28.573, 124.819, -178.462, 45.244, -179.734]
  Set speed (50.0 mm/s)
  MoveL 209 to (-36, 337.86, 0) mm, rotated rx 180 ry 0 rz 90 deg; joints [1.736, -27.348, 124.15, -178.477, 45.8, -179.713]
  MoveL 210 to (-36, 337.86, 20) mm, rotated rx 180 ry 0 rz 90 deg; joints [1.736, -28.573, 124.819, -178.462, 45.244, -179.734]
  Set speed (1000.0 mm/s)
  MoveL 211 to (-36, 287.09, 20) mm, rotated rx 180 ry 0 rz 90 deg; joints [1.664, -28.946, 122.58, -178.453, 42.632, -179.844]
  Set speed (50.0 mm/s)
  MoveL 212 to (-36, 287.09, 0) mm, rotated rx 180 ry 0 rz 90 deg; joints [1.664, -27.748, 121.929, -178.469, 43.179, -179.823]
  MoveL 213 to (-36, 287.09, 20) mm, rotated rx 180 ry 0 rz 90 deg; joints [1.664, -28.946, 122.58, -178.453, 42.632, -179.844]
  Set speed (1000.0 mm/s)
  MoveL 214 to (-36, 236.32, 20) mm, rotated rx -180 ry 0 rz 90 deg; joints [1.599, -29.175, 120.273, -178.438, 40.097, -179.952]
  Set speed (50.0 mm/s)
  MoveL 215 to (-36, 236.32, 0) mm, rotated rx 180 ry 0 rz 90 deg; joints [1.599, -28.003, 119.639, -178.455, 40.635, -179.93]
  MoveL 216 to (-36, 236.32, 20) mm, rotated rx -180 ry 0 rz 90 deg; joints [1.599, -29.175, 120.273, -178.438, 40.097, -179.952]
  Set speed (1000.0 mm/s)
  MoveL 217 to (-36, 185.55, 20) mm, rotated rx -180 ry 0 rz 90 deg; joints [1.538, -29.268, 117.899, -178.414, 37.631, -180.06]
  Set speed (50.0 mm/s)
  MoveL 218 to (-36, 185.55, 0) mm, rotated rx -180 ry 0 rz 90 deg; joints [1.538, -28.123, 117.281, -178.433, 38.158, -180.037]
  MoveL 219 to (-36, 185.55, 20) mm, rotated rx -180 ry 0 rz 90 deg; joints [1.538, -29.268, 117.899, -178.414, 37.631, -180.06]
  Set speed (1000.0 mm/s)
  MoveL 220 to (-77, 179.01, 20) mm, rotated rx -180 ry 0 rz 90 deg; joints [3.272, -29.272, 117.507, -176.597, 37.238, -180.166]
  Set speed (50.0 mm/s)
  MoveL 221 to (-77, 179.01, 0) mm, rotated rx 180 ry 0 rz 90 deg; joints [3.272, -28.131, 116.891, -176.638, 37.762, -180.116]
  MoveL 222 to (-77, 179.01, 20) mm, rotated rx -180 ry 0 rz 90 deg; joints [3.272, -29.272, 117.507, -176.597, 37.238, -180.166]
  Set speed (1000.0 mm/s)
  MoveL 223 to (-36, 134.78, 20) mm, rotated rx 180 ry 0 rz 90 deg; joints [1.482, -29.238, 115.461, -178.383, 35.225, -180.169]
  Set speed (50.0 mm/s)
  MoveL 224 to (-36, 134.78, 0) mm, rotated rx -180 ry 0 rz 90 deg; joints [1.482, -28.118, 114.856, -178.403, 35.739, -180.144]
  MoveL 225 to (-36, 134.78, 20) mm, rotated rx 180 ry 0 rz 90 deg; joints [1.482, -29.238, 115.461, -178.383, 35.225, -180.169]
  Set speed (1000.0 mm/s)
  MoveL 226 to (-36, 84.01, 20) mm, rotated rx -180 ry 0 rz 90 deg; joints [1.43, -29.09, 112.957, -178.342, 32.869, -180.282]
  Set speed (50.0 mm/s)
  MoveL 227 to (-36, 84.01, 0) mm, rotated rx 180 ry 0 rz 90 deg; joints [1.43, -27.997, 112.365, -178.364, 33.37, -180.255]
  MoveL 228 to (-36, 84.01, 20) mm, rotated rx -180 ry 0 rz 90 deg; joints [1.43, -29.09, 112.957, -178.342, 32.869, -180.282]
  Set speed (1000.0 mm/s)
  MoveL 229 to (-36, 33.24, 20) mm, rotated rx 180 ry 0 rz 90 deg; joints [1.382, -28.834, 110.387, -178.29, 30.557, -180.399]
  Set speed (50.0 mm/s)
  MoveL 230 to (-36, 33.24, 0) mm, rotated rx 180 ry 0 rz 90 deg; joints [1.382, -27.765, 109.807, -178.314, 31.044, -180.371]
  MoveL 231 to (-36, 33.24, 20) mm, rotated rx 180 ry 0 rz 90 deg; joints [1.382, -28.834, 110.387, -178.29, 30.557, -180.399]
  Set speed (1000.0 mm/s)
  MoveL 232 to (-36, -17.53, 20) mm, rotated rx -180 ry 0 rz 90 deg; joints [1.336, -28.474, 107.75, -178.225, 28.28, -180.525]
  Set speed (50.0 mm/s)
  MoveL 233 to (-36, -17.53, 0) mm, rotated rx -180 ry 0 rz 90 deg; joints [1.336, -27.429, 107.18, -178.252, 28.754, -180.494]
  MoveL 234 to (-36, -17.53, 20) mm, rotated rx -180 ry 0 rz 90 deg; joints [1.336, -28.474, 107.75, -178.225, 28.28, -180.525]
  Set speed (1000.0 mm/s)
  MoveL 235 to (-36, -68.3, 20) mm, rotated rx -180 ry 0 rz 90 deg; joints [1.294, -28.016, 105.045, -178.145, 26.033, -180.662]
  Set speed (50.0 mm/s)
  MoveL 236 to (-36, -68.3, 0) mm, rotated rx -180 ry 0 rz 90 deg; joints [1.294, -26.994, 104.483, -178.175, 26.493, -180.628]
  MoveL 237 to (-36, -68.3, 20) mm, rotated rx -180 ry 0 rz 90 deg; joints [1.294, -28.016, 105.045, -178.145, 26.033, -180.662]
  Set speed (1000.0 mm/s)
  MoveL 238 to (-36, -119.07, 20) mm, rotated rx -180 ry 0 rz 90 deg; joints [1.254, -27.465, 102.267, -178.045, 23.808, -180.814]
  Set speed (50.0 mm/s)
  MoveL 239 to (-36, -119.07, 0) mm, rotated rx 180 ry 0 rz 90 deg; joints [1.254, -26.464, 101.712, -178.079, 24.253, -180.777]
  MoveL 240 to (-36, -119.07, 20) mm, rotated rx -180 ry 0 rz 90 deg; joints [1.254, -27.465, 102.267, -178.045, 23.808, -180.814]
  Set speed (1000.0 mm/s)
  MoveL 241 to (-36, -169.84, 20) mm, rotated rx 180 ry 0 rz 90 deg; joints [1.216, -26.822, 99.414, -177.92, 21.598, -180.988]
  Set speed (50.0 mm/s)
  MoveL 242 to (-36, -169.84, 0) mm, rotated rx 180 ry 0 rz 90 deg; joints [1.216, -25.842, 98.866, -177.959, 22.03, -180.947]
  MoveL 243 to (-36, -169.84, 20) mm, rotated rx 180 ry 0 rz 90 deg; joints [1.216, -26.822, 99.414, -177.92, 21.598, -180.988]
  Set speed (1000.0 mm/s)
  MoveL 244 to (-36, -220.61, 20) mm, rotated rx 180 ry 0 rz 90 deg; joints [1.181, -26.091, 96.481, -177.762, 19.398, -181.193]
  Set speed (50.0 mm/s)
  MoveL 245 to (-36, -220.61, 0) mm, rotated rx -180 ry 0 rz 90 deg; joints [1.181, -25.13, 95.938, -177.807, 19.815, -181.145]
  MoveL 246 to (-36, -220.61, 20) mm, rotated rx 180 ry 0 rz 90 deg; joints [1.181, -26.091, 96.481, -177.762, 19.398, -181.193]
  Set speed (1000.0 mm/s)
  MoveL 247 to (-36, -271.37, 20) mm, rotated rx -180 ry 0 rz 90 deg; joints [1.147, -25.272, 93.464, -177.558, 17.201, -181.442]
  Set speed (50.0 mm/s)
  MoveL 248 to (-36, -271.37, 0) mm, rotated rx -180 ry 0 rz 90 deg; joints [1.147, -24.33, 92.923, -177.612, 17.602, -181.385]
  MoveL 249 to (-36, -271.37, 20) mm, rotated rx -180 ry 0 rz 90 deg; joints [1.147, -25.272, 93.464, -177.558, 17.201, -181.442]
  Set speed (1000.0 mm/s)
  MoveL 250 to (-36, -322.14, 20) mm, rotated rx 180 ry 0 rz 90 deg; joints [1.116, -24.365, 90.354, -177.285, 14.999, -181.755]
  Set speed (50.0 mm/s)
  MoveL 251 to (-36, -322.14, 0) mm, rotated rx -180 ry 0 rz 90 deg; joints [1.116, -23.44, 89.815, -177.352, 15.385, -181.686]
  MoveL 252 to (-36, -322.14, 20) mm, rotated rx 180 ry 0 rz 90 deg; joints [1.116, -24.365, 90.354, -177.285, 14.999, -181.755]
  Set speed (1000.0 mm/s)
  MoveL 253 to (-36, -372.91, 20) mm, rotated rx -180 ry 0 rz 90 deg; joints [1.086, -23.371, 87.143, -176.91, 12.786, -182.169]
  Set speed (50.0 mm/s)
  MoveL 254 to (-36, -372.91, 0) mm, rotated rx -180 ry 0 rz 90 deg; joints [1.086, -22.461, 86.605, -176.996, 13.157, -182.081]
  MoveL 255 to (-36, -372.91, 20) mm, rotated rx -180 ry 0 rz 90 deg; joints [1.086, -23.371, 87.143, -176.91, 12.786, -182.169]
  Set speed (1000.0 mm/s)
  MoveL 256 to (-77, -380.99, 20) mm, rotated rx 180 ry 0 rz 90 deg; joints [2.312, -23.179, 86.544, -173.224, 12.427, -184.822]
  Set speed (50.0 mm/s)
  MoveL 257 to (-77, -380.99, 0) mm, rotated rx 180 ry 0 rz 90 deg; joints [2.312, -22.272, 86.006, -173.416, 12.793, -184.625]
  MoveL 258 to (-77, -380.99, 20) mm, rotated rx 180 ry 0 rz 90 deg; joints [2.312, -23.179, 86.544, -173.224, 12.427, -184.822]
  Set speed (1000.0 mm/s)
  MoveL 259 to (-36, -423.68, 20) mm, rotated rx -180 ry 0 rz 90 deg; joints [1.058, -22.285, 83.823, -176.363, 10.554, -182.753]
  Set speed (50.0 mm/s)
  MoveL 260 to (-36, -423.68, 0) mm, rotated rx 180 ry 0 rz 90 deg; joints [1.058, -21.389, 83.283, -176.48, 10.909, -182.634]
  MoveL 261 to (-36, -423.68, 20) mm, rotated rx -180 ry 0 rz 90 deg; joints [1.058, -22.285, 83.823, -176.363, 10.554, -182.753]
  Set speed (1000.0 mm/s)
  MoveL 262 to (-36, -474.45, 20) mm, rotated rx 180 ry 0 rz 90 deg; joints [1.031, -21.106, 80.381, -175.499, 8.296, -183.653]
  Set speed (50.0 mm/s)
  MoveL 263 to (-36, -474.45, 0) mm, rotated rx -180 ry 0 rz 90 deg; joints [1.031, -20.222, 79.837, -175.674, 8.635, -183.476]
  MoveL 264 to (-36, -474.45, 20) mm, rotated rx 180 ry 0 rz 90 deg; joints [1.031, -21.106, 80.381, -175.499, 8.296, -183.653]
  Set speed (1000.0 mm/s)
  MoveL 265 to (-36, -525.22, 20) mm, rotated rx -180 ry 0 rz 90 deg; joints [1.005, -19.827, 76.801, -173.938, 6.003, -185.247]
  Set speed (50.0 mm/s)
  MoveL 266 to (-36, -525.22, 0) mm, rotated rx 180 ry 0 rz 90 deg; joints [1.005, -18.954, 76.252, -174.247, 6.325, -184.937]
  MoveL 267 to (-36, -525.22, 20) mm, rotated rx -180 ry 0 rz 90 deg; joints [1.005, -19.827, 76.801, -173.938, 6.003, -185.247]
  Set speed (1000.0 mm/s)
  MoveL 268 to (-36, -575.99, 20) mm, rotated rx 180 ry 0 rz 90 deg; joints [0.981, -18.441, 73.066, -170.313, 3.672, -188.905]
  Set speed (50.0 mm/s)
  MoveL 269 to (-36, -575.99, 0) mm, rotated rx 180 ry 0 rz 90 deg; joints [0.981, -17.578, 72.508, -171.054, 3.974, -188.162]
  MoveL 270 to (-36, -575.99, 20) mm, rotated rx 180 ry 0 rz 90 deg; joints [0.981, -18.441, 73.066, -170.313, 3.672, -188.905]
  Set speed (1000.0 mm/s)
  MoveL 271 to (40, -575.99, 20) mm, rotated rx -180 ry 0 rz 90 deg; joints [-1.09, -18.439, 73.06, -190.751, 3.68, -170.117]
  Set speed (50.0 mm/s)
  MoveL 272 to (40, -575.99, 0) mm, rotated rx 180 ry 0 rz 90 deg; joints [-1.09, -17.576, 72.502, -189.932, 3.981, -170.939]
  MoveL 273 to (40, -575.99, 20) mm, rotated rx -180 ry 0 rz 90 deg; joints [-1.09, -18.439, 73.06, -190.751, 3.68, -170.117]
  Set speed (1000.0 mm/s)
  MoveL 274 to (40, -525.82, 20) mm, rotated rx 180 ry 0 rz 90 deg; joints [-1.117, -19.809, 76.752, -186.763, 5.979, -174.142]
  Set speed (50.0 mm/s)
  MoveL 275 to (40, -525.82, 0) mm, rotated rx -180 ry 0 rz 90 deg; joints [-1.117, -18.937, 76.203, -186.418, 6.3, -174.488]
  MoveL 276 to (40, -525.82, 20) mm, rotated rx 180 ry 0 rz 90 deg; joints [-1.117, -19.809, 76.752, -186.763, 5.979, -174.142]
  Set speed (1000.0 mm/s)
  MoveL 277 to (40, -475.64, 20) mm, rotated rx 180 ry 0 rz 90 deg; joints [-1.145, -21.075, 80.293, -185.031, 8.244, -175.911]
  Set speed (50.0 mm/s)
  MoveL 278 to (40, -475.64, 0) mm, rotated rx 180 ry 0 rz 90 deg; joints [-1.145, -20.192, 79.75, -184.834, 8.582, -176.11]
  MoveL 279 to (40, -475.64, 20) mm, rotated rx 180 ry 0 rz 90 deg; joints [-1.145, -21.075, 80.293, -185.031, 8.244, -175.911]
  Set speed (1000.0 mm/s)
  MoveL 280 to (40, -425.47, 20) mm, rotated rx 180 ry 0 rz 90 deg; joints [-1.174, -22.243, 83.699, -184.068, 10.475, -176.912]
  Set speed (50.0 mm/s)
  MoveL 281 to (40, -425.47, 0) mm, rotated rx 180 ry 0 rz 90 deg; joints [-1.174, -21.348, 83.159, -183.936, 10.83, -177.047]
  MoveL 282 to (40, -425.47, 20) mm, rotated rx 180 ry 0 rz 90 deg; joints [-1.174, -22.243, 83.699, -184.068, 10.475, -176.912]
  Set speed (1000.0 mm/s)
  MoveL 283 to (0, -380.99, 20) mm, rotated rx -180 ry 0 rz 90 deg; joints [0, -23.211, 86.644, -180, 12.433, -180]
  Set speed (50.0 mm/s)
  MoveL 284 to (0, -380.99, 0) mm, rotated rx -180 ry 0 rz 90 deg; joints [0, -22.303, 86.106, -180, 12.803, -180]
  MoveL 285 to (0, -380.99, 20) mm, rotated rx -180 ry 0 rz 90 deg; joints [0, -23.211, 86.644, -180, 12.433, -180]
  Set speed (1000.0 mm/s)
  MoveL 286 to (40, -375.29, 20) mm, rotated rx -180 ry 0 rz 90 deg; joints [-1.205, -23.32, 86.985, -183.457, 12.681, -177.564]
  Set speed (50.0 mm/s)
  MoveL 287 to (40, -375.29, 0) mm, rotated rx 180 ry 0 rz 90 deg; joints [-1.205, -22.411, 86.447, -183.36, 13.051, -177.663]
  MoveL 288 to (40, -375.29, 20) mm, rotated rx -180 ry 0 rz 90 deg; joints [-1.205, -23.32, 86.985, -183.457, 12.681, -177.564]
  Set speed (1000.0 mm/s)
  MoveL 289 to (40, -325.12, 20) mm, rotated rx -180 ry 0 rz 90 deg; joints [-1.238, -24.308, 90.163, -183.037, 14.868, -178.026]
  Set speed (50.0 mm/s)
  MoveL 290 to (40, -325.12, 0) mm, rotated rx 180 ry 0 rz 90 deg; joints [-1.238, -23.384, 89.624, -182.962, 15.254, -178.104]
  MoveL 291 to (40, -325.12, 20) mm, rotated rx -180 ry 0 rz 90 deg; joints [-1.238, -24.308, 90.163, -183.037, 14.868, -178.026]
  Set speed (1000.0 mm/s)
  MoveL 292 to (40, -274.95, 20) mm, rotated rx 180 ry 0 rz 90 deg; joints [-1.272, -25.209, 93.242, -182.733, 17.044, -178.376]
  Set speed (50.0 mm/s)
  MoveL 293 to (40, -274.95, 0) mm, rotated rx -180 ry 0 rz 90 deg; joints [-1.272, -24.268, 92.702, -182.672, 17.445, -178.44]
  MoveL 294 to (40, -274.95, 20) mm, rotated rx 180 ry 0 rz 90 deg; joints [-1.272, -25.209, 93.242, -182.733, 17.044, -178.376]
  Set speed (1000.0 mm/s)
  MoveL 295 to (40, -224.77, 20) mm, rotated rx -180 ry 0 rz 90 deg; joints [-1.309, -26.026, 96.232, -182.503, 19.216, -178.653]
  Set speed (50.0 mm/s)
  MoveL 296 to (40, -224.77, 0) mm, rotated rx 180 ry 0 rz 90 deg; joints [-1.309, -25.067, 95.689, -182.452, 19.631, -178.707]
  MoveL 297 to (40, -224.77, 20) mm, rotated rx -180 ry 0 rz 90 deg; joints [-1.309, -26.026, 96.232, -182.503, 19.216, -178.653]
  Set speed (1000.0 mm/s)
  MoveL 298 to (40, -174.6, 20) mm, rotated rx 180 ry 0 rz 90 deg; joints [-1.347, -26.756, 99.137, -182.326, 21.39, -178.882]
  Set speed (50.0 mm/s)
  MoveL 299 to (40, -174.6, 0) mm, rotated rx 180 ry 0 rz 90 deg; joints [-1.347, -25.778, 98.589, -182.282, 21.819, -178.929]
  MoveL 300 to (40, -174.6, 20) mm, rotated rx 180 ry 0 rz 90 deg; joints [-1.347, -26.756, 99.137, -182.326, 21.39, -178.882]
  Set speed (1000.0 mm/s)
  MoveL 301 to (40, -124.43, 20) mm, rotated rx -180 ry 0 rz 90 deg; joints [-1.388, -27.4, 101.964, -182.185, 23.571, -179.076]
  Set speed (50.0 mm/s)
  MoveL 302 to (40, -124.43, 0) mm, rotated rx 180 ry 0 rz 90 deg; joints [-1.388, -26.402, 101.41, -182.147, 24.015, -179.118]
  MoveL 303 to (40, -124.43, 20) mm, rotated rx -180 ry 0 rz 90 deg; joints [-1.388, -27.4, 101.964, -182.185, 23.571, -179.076]
  Set speed (1000.0 mm/s)
  MoveL 304 to (40, -74.25, 20) mm, rotated rx -180 ry 0 rz 90 deg; joints [-1.432, -27.955, 104.718, -182.073, 25.768, -179.246]
  Set speed (50.0 mm/s)
  MoveL 305 to (40, -74.25, 0) mm, rotated rx 180 ry 0 rz 90 deg; joints [-1.432, -26.936, 104.157, -182.039, 26.226, -179.283]
  MoveL 306 to (40, -74.25, 20) mm, rotated rx -180 ry 0 rz 90 deg; joints [-1.432, -27.955, 104.718, -182.073, 25.768, -179.246]
  Set speed (1000.0 mm/s)
  MoveL 307 to (40, -24.08, 20) mm, rotated rx 180 ry 0 rz 90 deg; joints [-1.478, -28.42, 107.4, -181.983, 27.985, -179.398]
  Set speed (50.0 mm/s)
  MoveL 308 to (40, -24.08, 0) mm, rotated rx -180 ry 0 rz 90 deg; joints [-1.478, -27.378, 106.831, -181.952, 28.458, -179.432]
  MoveL 309 to (40, -24.08, 20) mm, rotated rx 180 ry 0 rz 90 deg; joints [-1.478, -28.42, 107.4, -181.983, 27.985, -179.398]
  Set speed (1000.0 mm/s)
  MoveL 310 to (40, 26.1, 20) mm, rotated rx -180 ry 0 rz 90 deg; joints [-1.528, -28.788, 110.015, -181.91, 30.231, -179.537]
  Set speed (50.0 mm/s)
  MoveL 311 to (40, 26.1, 0) mm, rotated rx 180 ry 0 rz 90 deg; joints [-1.528, -27.723, 109.436, -181.882, 30.716, -179.569]
  MoveL 312 to (40, 26.1, 20) mm, rotated rx -180 ry 0 rz 90 deg; joints [-1.528, -28.788, 110.015, -181.91, 30.231, -179.537]
  Set speed (1000.0 mm/s)
  MoveL 313 to (40, 76.27, 20) mm, rotated rx -180 ry 0 rz 90 deg; joints [-1.581, -29.057, 112.564, -181.851, 32.509, -179.667]
  Set speed (50.0 mm/s)
  MoveL 314 to (40, 76.27, 0) mm, rotated rx 180 ry 0 rz 90 deg; joints [-1.581, -27.968, 111.974, -181.826, 33.009, -179.697]
  MoveL 315 to (40, 76.27, 20) mm, rotated rx -180 ry 0 rz 90 deg; joints [-1.581, -29.057, 112.564, -181.851, 32.509, -179.667]
  Set speed (1000.0 mm/s)
  MoveL 316 to (40, 126.44, 20) mm, rotated rx 180 ry 0 rz 90 deg; joints [-1.637, -29.221, 115.049, -181.804, 34.83, -179.791]
  Set speed (50.0 mm/s)
  MoveL 317 to (40, 126.44, 0) mm, rotated rx -180 ry 0 rz 90 deg; joints [-1.637, -28.106, 114.446, -181.781, 35.342, -179.819]
  MoveL 318 to (40, 126.44, 20) mm, rotated rx 180 ry 0 rz 90 deg; joints [-1.637, -29.221, 115.049, -181.804, 34.83, -179.791]
  Set speed (1000.0 mm/s)
  MoveL 319 to (40, 176.62, 20) mm, rotated rx 180 ry 0 rz 90 deg; joints [-1.698, -29.272, 117.47, -181.768, 37.199, -179.912]
  Set speed (50.0 mm/s)
  MoveL 320 to (40, 176.62, 0) mm, rotated rx -180 ry 0 rz 90 deg; joints [-1.698, -28.131, 116.854, -181.747, 37.723, -179.938]
  MoveL 321 to (40, 176.62, 20) mm, rotated rx 180 ry 0 rz 90 deg; joints [-1.698, -29.272, 117.47, -181.768, 37.199, -179.912]
  Set speed (1000.0 mm/s)
  MoveL 322 to (0, 179.01, 20) mm, rotated rx -180 ry 0 rz 90 deg; joints [0, -29.271, 117.612, -180, 37.341, -180]
  Set speed (50.0 mm/s)
  MoveL 323 to (0, 179.01, 0) mm, rotated rx -180 ry 0 rz 90 deg; joints [0, -28.129, 116.995, -180, 37.866, -180]
  MoveL 324 to (0, 179.01, 20) mm, rotated rx -180 ry 0 rz 90 deg; joints [0, -29.271, 117.612, -180, 37.341, -180]
  Set speed (1000.0 mm/s)
  MoveL 325 to (40, 226.79, 20) mm, rotated rx -180 ry 0 rz 90 deg; joints [-1.764, -29.203, 119.827, -181.74, 39.624, -180.03]
  Set speed (50.0 mm/s)
  MoveL 326 to (40, 226.79, 0) mm, rotated rx -180 ry 0 rz 90 deg; joints [-1.764, -28.036, 119.196, -181.721, 40.16, -180.055]
  MoveL 327 to (40, 226.79, 20) mm, rotated rx -180 ry 0 rz 90 deg; joints [-1.764, -29.203, 119.827, -181.74, 39.624, -180.03]
  Set speed (1000.0 mm/s)
  MoveL 328 to (40, 327.14, 20) mm, rotated rx -180 ry 0 rz 90 deg; joints [-1.911, -28.665, 124.346, -181.71, 44.678, -180.269]
  Set speed (50.0 mm/s)
  MoveL 329 to (40, 327.14, 0) mm, rotated rx -180 ry 0 rz 90 deg; joints [-1.911, -27.446, 123.681, -181.694, 45.232, -180.292]
  MoveL 330 to (40, 327.14, 20) mm, rotated rx -180 ry 0 rz 90 deg; joints [-1.911, -28.665, 124.346, -181.71, 44.678, -180.269]
  Set speed (1000.0 mm/s)
  MoveL 331 to (40, 377.31, 20) mm, rotated rx -180 ry 0 rz 90 deg; joints [-1.994, -28.176, 126.505, -181.707, 47.325, -180.393]
  Set speed (50.0 mm/s)
  MoveL 332 to (40, 377.31, 0) mm, rotated rx 180 ry 0 rz 90 deg; joints [-1.994, -26.931, 125.821, -181.692, 47.886, -180.415]
  MoveL 333 to (40, 377.31, 20) mm, rotated rx -180 ry 0 rz 90 deg; joints [-1.994, -28.176, 126.505, -181.707, 47.325, -180.393]
  Set speed (1000.0 mm/s)
  MoveL 334 to (40, 427.49, 20) mm, rotated rx 180 ry 0 rz 90 deg; joints [-2.085, -27.521, 128.593, -181.712, 50.066, -180.522]
  Set speed (50.0 mm/s)
  MoveL 335 to (40, 427.49, 0) mm, rotated rx 180 ry 0 rz 90 deg; joints [-2.085, -26.252, 127.889, -181.698, 50.631, -180.544]
  MoveL 336 to (40, 427.49, 20) mm, rotated rx 180 ry 0 rz 90 deg; joints [-2.085, -27.521, 128.593, -181.712, 50.066, -180.522]
  Set speed (1000.0 mm/s)
  MoveL 337 to (0, 459.01, 20) mm, rotated rx 180 ry 0 rz 90 deg; joints [0, -27.007, 129.897, -180, 51.89, -180]
  Set speed (50.0 mm/s)
  MoveL 338 to (0, 459.01, 0) mm, rotated rx 180 ry 0 rz 90 deg; joints [0, -25.723, 129.179, -180, 52.456, -180]
  MoveL 339 to (0, 459.01, 20) mm, rotated rx 180 ry 0 rz 90 deg; joints [0, -27.007, 129.897, -180, 51.89, -180]
  Set speed (1000.0 mm/s)
  MoveL 340 to (40, 477.66, 20) mm, rotated rx -180 ry 0 rz 90 deg; joints [-2.185, -26.688, 130.606, -181.724, 52.91, -180.659]
  Set speed (50.0 mm/s)
  MoveL 341 to (40, 477.66, 0) mm, rotated rx -180 ry 0 rz 90 deg; joints [-2.185, -25.396, 129.88, -181.711, 53.476, -180.68]
  MoveL 342 to (40, 477.66, 20) mm, rotated rx -180 ry 0 rz 90 deg; joints [-2.185, -26.688, 130.606, -181.724, 52.91, -180.659]
  Set speed (1000.0 mm/s)
  MoveL 343 to (40, 527.84, 20) mm, rotated rx -180 ry 0 rz 90 deg; joints [-2.295, -25.66, 132.541, -181.745, 55.87, -180.805]
  Set speed (50.0 mm/s)
  MoveL 344 to (40, 527.84, 0) mm, rotated rx 180 ry 0 rz 90 deg; joints [-2.295, -24.349, 131.791, -181.733, 56.432, -180.825]
  MoveL 345 to (40, 527.84, 20) mm, rotated rx -180 ry 0 rz 90 deg; joints [-2.295, -25.66, 132.541, -181.745, 55.87, -180.805]
  Set speed (1000.0 mm/s)
  MoveL 346 to (40, 578.01, 20) mm, rotated rx 180 ry 0 rz 90 deg; joints [-2.416, -24.421, 134.389, -181.775, 58.956, -180.963]
  Set speed (50.0 mm/s)
  MoveL 347 to (40, 578.01, 0) mm, rotated rx 180 ry 0 rz 90 deg; joints [-2.416, -23.094, 133.615, -181.764, 59.508, -180.983]
  MoveL 348 to (40, 578.01, 20) mm, rotated rx 180 ry 0 rz 90 deg; joints [-2.416, -24.421, 134.389, -181.775, 58.956, -180.963]
  Set speed (1000.0 mm/s)
  MoveL 349 to (11, 578.01, 20) mm, rotated rx 180 ry 0 rz 90 deg; joints [-0.665, -24.4, 134.418, -180.488, 59.016, -180.265]
  Set speed (50.0 mm/s)
  MoveL 350 to (11, 578.01, 0) mm, rotated rx 180 ry 0 rz 90 deg; joints [-0.665, -23.073, 133.643, -180.485, 59.569, -180.271]
  MoveL 351 to (11, 578.01, 20) mm, rotated rx 180 ry 0 rz 90 deg; joints [-0.665, -24.4, 134.418, -180.488, 59.016, -180.265]
  Set speed (1000.0 mm/s)
  MoveL 352 to (11, 613.01, 20) mm, rotated rx -180 ry 0 rz 90 deg; joints [-0.69, -23.397, 135.653, -180.495, 61.255, -180.298]
  Set speed (50.0 mm/s)
  MoveL 353 to (11, 613.01, 0) mm, rotated rx -180 ry 0 rz 90 deg; joints [-0.69, -22.062, 134.861, -180.493, 61.798, -180.304]
  MoveL 354 to (11, 613.01, 20) mm, rotated rx -180 ry 0 rz 90 deg; joints [-0.69, -23.397, 135.653, -180.495, 61.255, -180.298]
  Set speed (1000.0 mm/s)
  MoveL 355 to (11, 648.01, 20) mm, rotated rx 180 ry 0 rz 90 deg; joints [-0.718, -22.277, 136.842, -180.505, 63.564, -180.333]
  Set speed (50.0 mm/s)
  MoveL 356 to (11, 648.01, 0) mm, rotated rx 180 ry 0 rz 90 deg; joints [-0.718, -20.937, 136.032, -180.502, 64.093, -180.338]
  MoveL 357 to (11, 648.01, 20) mm, rotated rx 180 ry 0 rz 90 deg; joints [-0.718, -22.277, 136.842, -180.505, 63.564, -180.333]
  Set speed (1000.0 mm/s)
  MoveL 358 to (11, 683.01, 20) mm, rotated rx -180 ry 0 rz 90 deg; joints [-0.748, -21.031, 137.981, -180.515, 65.948, -180.371]
  Set speed (50.0 mm/s)
  MoveL 359 to (11, 683.01, 0) mm, rotated rx -180 ry 0 rz 90 deg; joints [-0.748, -19.691, 137.152, -180.513, 66.459, -180.376]
  MoveL 360 to (11, 683.01, 20) mm, rotated rx -180 ry 0 rz 90 deg; joints [-0.748, -21.031, 137.981, -180.515, 65.948, -180.371]
  Set speed (1000.0 mm/s)
  MoveL 361 to (11, 718.01, 20) mm, rotated rx 180 ry 0 rz 90 deg; joints [-0.78, -19.656, 139.066, -180.528, 68.408, -180.412]
  Set speed (50.0 mm/s)
  MoveL 362 to (11, 718.01, 0) mm, rotated rx -180 ry 0 rz 90 deg; joints [-0.78, -18.319, 138.218, -180.526, 68.897, -180.417]
  MoveL 363 to (11, 718.01, 20) mm, rotated rx 180 ry 0 rz 90 deg; joints [-0.78, -19.656, 139.066, -180.528, 68.408, -180.412]
  Set speed (1000.0 mm/s)
  MoveL 364 to (65.2, 688.01, 20) mm, rotated rx -180 ry 0 rz 90 deg; joints [-4.449, -20.936, 138.061, -183.062, 66.071, -182.218]
  Set speed (50.0 mm/s)
  MoveL 365 to (65.2, 688.01, 0) mm, rotated rx -180 ry 0 rz 90 deg; joints [-4.449, -19.596, 137.231, -183.05, 66.58, -182.247]
  MoveL 366 to (65.2, 688.01, 20) mm, rotated rx -180 ry 0 rz 90 deg; joints [-4.449, -20.936, 138.061, -183.062, 66.071, -182.218]
  Set speed (1000.0 mm/s)
  MoveL 367 to (65.2, 651.34, 20) mm, rotated rx 180 ry 0 rz 90 deg; joints [-4.263, -22.244, 136.874, -182.994, 63.584, -181.983]
  Set speed (50.0 mm/s)
  MoveL 368 to (65.2, 651.34, 0) mm, rotated rx -180 ry 0 rz 90 deg; joints [-4.263, -20.904, 136.064, -182.981, 64.112, -182.013]
  MoveL 369 to (65.2, 651.34, 20) mm, rotated rx 180 ry 0 rz 90 deg; joints [-4.263, -22.244, 136.874, -182.994, 63.584, -181.983]
  Set speed (1000.0 mm/s)
  MoveL 370 to (65.2, 614.68, 20) mm, rotated rx -180 ry 0 rz 90 deg; joints [-4.092, -23.415, 135.633, -182.938, 61.178, -181.765]
  Set speed (50.0 mm/s)
  MoveL 371 to (65.2, 614.68, 0) mm, rotated rx 180 ry 0 rz 90 deg; joints [-4.092, -22.08, 134.841, -182.923, 61.72, -181.797]
  MoveL 372 to (65.2, 614.68, 20) mm, rotated rx -180 ry 0 rz 90 deg; joints [-4.092, -23.415, 135.633, -182.938, 61.178, -181.765]
  Set speed (1000.0 mm/s)
  MoveL 373 to (65.2, 578.01, 20) mm, rotated rx -180 ry 0 rz 90 deg; joints [-3.935, -24.459, 134.339, -182.892, 58.847, -181.562]
  Set speed (50.0 mm/s)
  MoveL 374 to (65.2, 578.01, 0) mm, rotated rx 180 ry 0 rz 90 deg; joints [-3.935, -23.132, 133.566, -182.876, 59.399, -181.595]
  MoveL 375 to (65.2, 578.01, 20) mm, rotated rx -180 ry 0 rz 90 deg; joints [-3.935, -24.459, 134.339, -182.892, 58.847, -181.562]
  Set speed (1000.0 mm/s)
  MoveL 376 to (114, 657.41, 20) mm, rotated rx 180 ry 0 rz 90 deg; joints [-7.478, -22.208, 136.909, -185.248, 63.558, -183.482]
  Set speed (50.0 mm/s)
  MoveL 377 to (114, 657.41, 0) mm, rotated rx -180 ry 0 rz 90 deg; joints [-7.478, -20.868, 136.098, -185.224, 64.084, -183.536]
  MoveL 378 to (114, 657.41, 20) mm, rotated rx 180 ry 0 rz 90 deg; joints [-7.478, -22.208, 136.909, -185.248, 63.558, -183.482]
  Set speed (1000.0 mm/s)
  MoveL 379 to (114, 608.07, 20) mm, rotated rx -180 ry 0 rz 90 deg; joints [-7.08, -23.752, 135.237, -185.12, 60.37, -182.977]
  Set speed (50.0 mm/s)
  MoveL 380 to (114, 608.07, 0) mm, rotated rx -180 ry 0 rz 90 deg; joints [-7.08, -22.419, 134.451, -185.092, 60.914, -183.033]
  MoveL 381 to (114, 608.07, 20) mm, rotated rx -180 ry 0 rz 90 deg; joints [-7.08, -23.752, 135.237, -185.12, 60.37, -182.977]
  Set speed (1000.0 mm/s)
  MoveL 382 to (114, 558.74, 20) mm, rotated rx -180 ry 0 rz 90 deg; joints [-6.722, -25.07, 133.474, -185.021, 57.311, -182.517]
  Set speed (50.0 mm/s)
  MoveL 383 to (114, 558.74, 0) mm, rotated rx 180 ry 0 rz 90 deg; joints [-6.722, -23.75, 132.712, -184.991, 57.867, -182.574]
  MoveL 384 to (114, 558.74, 20) mm, rotated rx -180 ry 0 rz 90 deg; joints [-6.722, -25.07, 133.474, -185.021, 57.311, -182.517]
  Set speed (1000.0 mm/s)
  MoveL 385 to (114, 509.4, 20) mm, rotated rx 180 ry 0 rz 90 deg; joints [-6.399, -26.178, 131.625, -184.95, 54.373, -182.093]
  Set speed (50.0 mm/s)
  MoveL 386 to (114, 509.4, 0) mm, rotated rx -180 ry 0 rz 90 deg; joints [-6.399, -24.875, 130.886, -184.916, 54.935, -182.152]
  MoveL 387 to (114, 509.4, 20) mm, rotated rx 180 ry 0 rz 90 deg; joints [-6.399, -26.178, 131.625, -184.95, 54.373, -182.093]
  Set speed (1000.0 mm/s)
  MoveL 388 to (72, 459.01, 20) mm, rotated rx 180 ry 0 rz 90 deg; joints [-3.861, -27.048, 129.8, -183.094, 51.729, -181.085]
  Set speed (50.0 mm/s)
  MoveL 389 to (72, 459.01, 0) mm, rotated rx -180 ry 0 rz 90 deg; joints [-3.861, -25.765, 129.083, -183.07, 52.294, -181.123]
  MoveL 390 to (72, 459.01, 20) mm, rotated rx 180 ry 0 rz 90 deg; joints [-3.861, -27.048, 129.8, -183.094, 51.729, -181.085]
  Set speed (1000.0 mm/s)
  MoveL 391 to (114, 460.07, 20) mm, rotated rx -180 ry 0 rz 90 deg; joints [-6.105, -27.092, 129.696, -184.903, 51.547, -181.698]
  Set speed (50.0 mm/s)
  MoveL 392 to (114, 460.07, 0) mm, rotated rx 180 ry 0 rz 90 deg; joints [-6.105, -25.81, 128.98, -184.865, 52.111, -181.759]
  MoveL 393 to (114, 460.07, 20) mm, rotated rx -180 ry 0 rz 90 deg; joints [-6.105, -27.092, 129.696, -184.903, 51.547, -181.698]
  Set speed (1000.0 mm/s)
  MoveL 394 to (147, 459.01, 20) mm, rotated rx 180 ry 0 rz 90 deg; joints [-7.845, -27.176, 129.493, -186.326, 51.225, -182.14]
  Set speed (50.0 mm/s)
  MoveL 395 to (147, 459.01, 0) mm, rotated rx 180 ry 0 rz 90 deg; joints [-7.845, -25.896, 128.779, -186.276, 51.787, -182.22]
  MoveL 396 to (147, 459.01, 20) mm, rotated rx 180 ry 0 rz 90 deg; joints [-7.845, -27.176, 129.493, -186.326, 51.225, -182.14]
  Set speed (1000.0 mm/s)
  MoveL 397 to (114, 410.73, 20) mm, rotated rx -180 ry 0 rz 90 deg; joints [-5.837, -27.828, 127.693, -184.878, 48.822, -181.326]
  Set speed (50.0 mm/s)
  MoveL 398 to (114, 410.73, 0) mm, rotated rx -180 ry 0 rz 90 deg; joints [-5.837, -26.568, 126.997, -184.836, 49.384, -181.39]
  MoveL 399 to (114, 410.73, 20) mm, rotated rx -180 ry 0 rz 90 deg; joints [-5.837, -27.828, 127.693, -184.878, 48.822, -181.326]
  Set speed (1000.0 mm/s)
  MoveL 400 to (114, 361.39, 20) mm, rotated rx -180 ry 0 rz 90 deg; joints [-5.591, -28.398, 125.618, -184.874, 46.19, -180.972]
  Set speed (50.0 mm/s)
  MoveL 401 to (114, 361.39, 0) mm, rotated rx 180 ry 0 rz 90 deg; joints [-5.591, -27.163, 124.942, -184.829, 46.747, -181.037]
  MoveL 402 to (114, 361.39, 20) mm, rotated rx -180 ry 0 rz 90 deg; joints [-5.591, -28.398, 125.618, -184.874, 46.19, -180.972]
  Set speed (1000.0 mm/s)
  MoveL 403 to (114, 312.06, 20) mm, rotated rx -180 ry 0 rz 90 deg; joints [-5.365, -28.816, 123.477, -184.891, 43.642, -180.631]
  Set speed (50.0 mm/s)
  MoveL 404 to (114, 312.06, 0) mm, rotated rx -180 ry 0 rz 90 deg; joints [-5.365, -27.607, 122.819, -184.842, 44.192, -180.698]
  MoveL 405 to (114, 312.06, 20) mm, rotated rx -180 ry 0 rz 90 deg; joints [-5.365, -28.816, 123.477, -184.891, 43.642, -180.631]
  Set speed (1000.0 mm/s)
  MoveL 406 to (114, 262.72, 20) mm, rotated rx -180 ry 0 rz 90 deg; joints [-5.157, -29.094, 121.27, -184.929, 41.168, -180.297]
  Set speed (50.0 mm/s)
  MoveL 407 to (114, 262.72, 0) mm, rotated rx 180 ry 0 rz 90 deg; joints [-5.157, -27.91, 120.629, -184.877, 41.708, -180.367]
  MoveL 408 to (114, 262.72, 20) mm, rotated rx -180 ry 0 rz 90 deg; joints [-5.157, -29.094, 121.27, -184.929, 41.168, -180.297]
  Set speed (1000.0 mm/s)
  MoveL 409 to (114, 213.39, 20) mm, rotated rx -180 ry 0 rz 90 deg; joints [-4.964, -29.241, 119.001, -184.99, 38.76, -179.967]
  Set speed (50.0 mm/s)
  MoveL 410 to (114, 213.39, 0) mm, rotated rx -180 ry 0 rz 90 deg; joints [-4.964, -28.084, 118.375, -184.933, 39.29, -180.04]
  MoveL 411 to (114, 213.39, 20) mm, rotated rx -180 ry 0 rz 90 deg; joints [-4.964, -29.241, 119.001, -184.99, 38.76, -179.967]
  Set speed (1000.0 mm/s)
  MoveL 412 to (40, 276.97, 20) mm, rotated rx 180 ry 0 rz 90 deg; joints [-1.834, -29.004, 122.12, -181.721, 42.114, -180.149]
  Set speed (50.0 mm/s)
  MoveL 413 to (40, 276.97, 0) mm, rotated rx -180 ry 0 rz 90 deg; joints [-1.834, -27.811, 121.472, -181.703, 42.66, -180.173]
  MoveL 414 to (40, 276.97, 20) mm, rotated rx 180 ry 0 rz 90 deg; joints [-1.834, -29.004, 122.12, -181.721, 42.114, -180.149]
  Set speed (1000.0 mm/s)
  MoveL 415 to (72, 179.01, 20) mm, rotated rx -180 ry 0 rz 90 deg; joints [-3.06, -29.272, 117.52, -183.181, 37.251, -179.846]
  Set speed (50.0 mm/s)
  MoveL 416 to (72, 179.01, 0) mm, rotated rx -180 ry 0 rz 90 deg; joints [-3.06, -28.131, 116.904, -183.144, 37.775, -179.893]
  MoveL 417 to (72, 179.01, 20) mm, rotated rx -180 ry 0 rz 90 deg; joints [-3.06, -29.272, 117.52, -183.181, 37.251, -179.846]
  Set speed (1000.0 mm/s)
  MoveL 418 to (114, 164.05, 20) mm, rotated rx 180 ry 0 rz 90 deg; joints [-4.785, -29.268, 116.669, -185.074, 36.411, -179.635]
  Set speed (50.0 mm/s)
  MoveL 419 to (114, 164.05, 0) mm, rotated rx 180 ry 0 rz 90 deg; joints [-4.785, -28.136, 116.057, -185.012, 36.929, -179.712]
  MoveL 420 to (114, 164.05, 20) mm, rotated rx 180 ry 0 rz 90 deg; joints [-4.785, -29.268, 116.669, -185.074, 36.411, -179.635]
  Set speed (1000.0 mm/s)
  MoveL 421 to (147, 179.01, 20) mm, rotated rx -180 ry 0 rz 90 deg; joints [-6.228, -29.272, 117.23, -186.519, 36.971, -179.632]
  Set speed (50.0 mm/s)
  MoveL 422 to (147, 179.01, 0) mm, rotated rx -180 ry 0 rz 90 deg; joints [-6.228, -28.134, 116.616, -186.441, 37.491, -179.729]
  MoveL 423 to (147, 179.01, 20) mm, rotated rx -180 ry 0 rz 90 deg; joints [-6.228, -29.272, 117.23, -186.519, 36.971, -179.632]
  Set speed (1000.0 mm/s)
  MoveL 424 to (114, 114.71, 20) mm, rotated rx 180 ry 0 rz 90 deg; joints [-4.618, -29.181, 114.275, -185.184, 34.111, -179.296]
  Set speed (50.0 mm/s)
  MoveL 425 to (114, 114.71, 0) mm, rotated rx -180 ry 0 rz 90 deg; joints [-4.618, -28.074, 113.676, -185.117, 34.618, -179.377]
  MoveL 426 to (114, 114.71, 20) mm, rotated rx 180 ry 0 rz 90 deg; joints [-4.618, -29.181, 114.275, -185.184, 34.111, -179.296]
  Set speed (1000.0 mm/s)
  MoveL 427 to (114, 65.38, 20) mm, rotated rx 180 ry 0 rz 90 deg; joints [-4.463, -28.989, 111.82, -185.324, 31.857, -178.946]
  Set speed (50.0 mm/s)
  MoveL 428 to (114, 65.38, 0) mm, rotated rx 180 ry 0 rz 90 deg; joints [-4.463, -27.907, 111.233, -185.251, 32.35, -179.032]
  MoveL 429 to (114, 65.38, 20) mm, rotated rx 180 ry 0 rz 90 deg; joints [-4.463, -28.989, 111.82, -185.324, 31.857, -178.946]
  Set speed (1000.0 mm/s)
  MoveL 430 to (114, 16.04, 20) mm, rotated rx -180 ry 0 rz 90 deg; joints [-4.318, -28.697, 109.301, -185.498, 29.638, -178.576]
  Set speed (50.0 mm/s)
  MoveL 431 to (114, 16.04, 0) mm, rotated rx 180 ry 0 rz 90 deg; joints [-4.318, -27.638, 108.725, -185.418, 30.119, -178.668]
  MoveL 432 to (114, 16.04, 20) mm, rotated rx -180 ry 0 rz 90 deg; joints [-4.318, -28.697, 109.301, -185.498, 29.638, -178.576]
  Set speed (1000.0 mm/s)
  MoveL 433 to (114, -33.29, 20) mm, rotated rx -180 ry 0 rz 90 deg; joints [-4.182, -28.309, 106.719, -185.713, 27.451, -178.179]
  Set speed (50.0 mm/s)
  MoveL 434 to (114, -33.29, 0) mm, rotated rx -180 ry 0 rz 90 deg; joints [-4.182, -27.273, 106.152, -185.625, 27.918, -178.279]
  MoveL 435 to (114, -33.29, 20) mm, rotated rx -180 ry 0 rz 90 deg; joints [-4.182, -28.309, 106.719, -185.713, 27.451, -178.179]
  Set speed (1000.0 mm/s)
  MoveL 436 to (114, -82.63, 20) mm, rotated rx -180 ry 0 rz 90 deg; joints [-4.054, -27.832, 104.07, -185.978, 25.289, -177.744]
  Set speed (50.0 mm/s)
  MoveL 437 to (114, -82.63, 0) mm, rotated rx 180 ry 0 rz 90 deg; joints [-4.054, -26.817, 103.511, -185.879, 25.741, -177.853]
  MoveL 438 to (114, -82.63, 20) mm, rotated rx -180 ry 0 rz 90 deg; joints [-4.054, -27.832, 104.07, -185.978, 25.289, -177.744]
  Set speed (1000.0 mm/s)
  MoveL 439 to (114, -131.97, 20) mm, rotated rx 180 ry 0 rz 90 deg; joints [-3.934, -27.267, 101.352, -186.306, 23.145, -177.257]
  Set speed (50.0 mm/s)
  MoveL 440 to (114, -131.97, 0) mm, rotated rx 180 ry 0 rz 90 deg; joints [-3.934, -26.273, 100.8, -186.194, 23.584, -177.378]
  MoveL 441 to (114, -131.97, 20) mm, rotated rx 180 ry 0 rz 90 deg; joints [-3.934, -27.267, 101.352, -186.306, 23.145, -177.257]
  Set speed (1000.0 mm/s)
  MoveL 442 to (114, -181.3, 20) mm, rotated rx -180 ry 0 rz 90 deg; joints [-3.82, -26.617, 98.563, -186.714, 21.015, -176.699]
  Set speed (50.0 mm/s)
  MoveL 443 to (114, -181.3, 0) mm, rotated rx -180 ry 0 rz 90 deg; joints [-3.82, -25.643, 98.016, -186.587, 21.439, -176.836]
  MoveL 444 to (114, -181.3, 20) mm, rotated rx -180 ry 0 rz 90 deg; joints [-3.82, -26.617, 98.563, -186.714, 21.015, -176.699]
  Set speed (1000.0 mm/s)
  MoveL 445 to (114, -230.64, 20) mm, rotated rx -180 ry 0 rz 90 deg; joints [-3.713, -25.884, 95.696, -187.231, 18.893, -176.042]
  Set speed (50.0 mm/s)
  MoveL 446 to (114, -230.64, 0) mm, rotated rx -180 ry 0 rz 90 deg; joints [-3.713, -24.928, 95.153, -187.082, 19.302, -176.199]
  MoveL 447 to (114, -230.64, 20) mm, rotated rx -180 ry 0 rz 90 deg; joints [-3.713, -25.884, 95.696, -187.231, 18.893, -176.042]
  Set speed (1000.0 mm/s)
  MoveL 448 to (114, -279.97, 20) mm, rotated rx 180 ry 0 rz 90 deg; joints [-3.612, -25.068, 92.747, -187.897, 16.773, -175.244]
  Set speed (50.0 mm/s)
  MoveL 449 to (114, -279.97, 0) mm, rotated rx -180 ry 0 rz 90 deg; joints [-3.612, -24.13, 92.207, -187.719, 17.168, -175.429]
  MoveL 450 to (114, -279.97, 20) mm, rotated rx 180 ry 0 rz 90 deg; joints [-3.612, -25.068, 92.747, -187.897, 16.773, -175.244]
  Set speed (1000.0 mm/s)
  MoveL 451 to (114, -329.31, 20) mm, rotated rx -180 ry 0 rz 90 deg; joints [-3.516, -24.17, 89.709, -188.778, 14.651, -174.237]
  Set speed (50.0 mm/s)
  MoveL 452 to (114, -329.31, 0) mm, rotated rx 180 ry 0 rz 90 deg; joints [-3.516, -23.248, 89.171, -188.56, 15.03, -174.463]
  MoveL 453 to (114, -329.31, 20) mm, rotated rx -180 ry 0 rz 90 deg; joints [-3.516, -24.17, 89.709, -188.778, 14.651, -174.237]
  Set speed (1000.0 mm/s)
  MoveL 454 to (72, -380.99, 20) mm, rotated rx -180 ry 0 rz 90 deg; joints [-2.162, -23.183, 86.557, -186.335, 12.427, -175.493]
  Set speed (50.0 mm/s)
  MoveL 455 to (72, -380.99, 0) mm, rotated rx 180 ry 0 rz 90 deg; joints [-2.162, -22.276, 86.018, -186.155, 12.794, -175.677]
  MoveL 456 to (72, -380.99, 20) mm, rotated rx -180 ry 0 rz 90 deg; joints [-2.162, -23.183, 86.557, -186.335, 12.427, -175.493]
  Set speed (1000.0 mm/s)
  MoveL 457 to (114, -378.65, 20) mm, rotated rx -180 ry 0 rz 90 deg; joints [-3.425, -23.189, 86.575, -189.988, 12.52, -172.908]
  Set speed (50.0 mm/s)
  MoveL 458 to (114, -378.65, 0) mm, rotated rx 180 ry 0 rz 90 deg; joints [-3.425, -22.281, 86.037, -189.708, 12.884, -173.195]
  MoveL 459 to (114, -378.65, 20) mm, rotated rx -180 ry 0 rz 90 deg; joints [-3.425, -23.189, 86.575, -189.988, 12.52, -172.908]
  Set speed (1000.0 mm/s)
  MoveL 460 to (147, -380.99, 20) mm, rotated rx -180 ry 0 rz 90 deg; joints [-4.408, -23.093, 86.278, -193.006, 12.411, -170.716]
  Set speed (50.0 mm/s)
  MoveL 461 to (147, -380.99, 0) mm, rotated rx -180 ry 0 rz 90 deg; joints [-4.408, -22.187, 85.74, -192.641, 12.769, -171.091]
  MoveL 462 to (147, -380.99, 20) mm, rotated rx -180 ry 0 rz 90 deg; joints [-4.408, -23.093, 86.278, -193.006, 12.411, -170.716]
  Set speed (1000.0 mm/s)
  MoveL 463 to (114, -427.98, 20) mm, rotated rx -180 ry 0 rz 90 deg; joints [-3.339, -22.122, 83.336, -191.739, 10.38, -171.044]
  Set speed (50.0 mm/s)
  MoveL 464 to (114, -427.98, 0) mm, rotated rx -180 ry 0 rz 90 deg; joints [-3.339, -21.228, 82.796, -191.358, 10.726, -171.431]
  MoveL 465 to (114, -427.98, 20) mm, rotated rx -180 ry 0 rz 90 deg; joints [-3.339, -22.122, 83.336, -191.739, 10.38, -171.044]
  Set speed (1000.0 mm/s)
  MoveL 466 to (114, -477.32, 20) mm, rotated rx -180 ry 0 rz 90 deg; joints [-3.257, -20.965, 79.98, -194.47, 8.227, -168.205]
  Set speed (50.0 mm/s)
  MoveL 467 to (114, -477.32, 0) mm, rotated rx 180 ry 0 rz 90 deg; joints [-3.257, -20.083, 79.436, -193.908, 8.555, -168.773]
  MoveL 468 to (114, -477.32, 20) mm, rotated rx -180 ry 0 rz 90 deg; joints [-3.257, -20.965, 79.98, -194.47, 8.227, -168.205]
  Set speed (1000.0 mm/s)
  MoveL 469 to (114, -526.65, 20) mm, rotated rx -180 ry 0 rz 90 deg; joints [-3.179, -19.714, 76.492, -199.262, 6.073, -163.31]
  Set speed (50.0 mm/s)
  MoveL 470 to (114, -526.65, 0) mm, rotated rx -180 ry 0 rz 90 deg; joints [-3.179, -18.843, 75.943, -198.312, 6.377, -164.266]
  MoveL 471 to (114, -526.65, 20) mm, rotated rx -180 ry 0 rz 90 deg; joints [-3.179, -19.714, 76.492, -199.262, 6.073, -163.31]
  Set speed (1000.0 mm/s)
  MoveL 472 to (114, -575.99, 20) mm, rotated rx -180 ry 0 rz 90 deg; joints [-3.104, -18.362, 72.856, -209.521, 3.966, -152.952]
  Set speed (50.0 mm/s)
  MoveL 473 to (114, -575.99, 0) mm, rotated rx -180 ry 0 rz 90 deg; joints [-3.104, -17.499, 72.298, -207.491, 4.234, -154.987]
  MoveL 474 to (114, -575.99, 20) mm, rotated rx -180 ry 0 rz 90 deg; joints [-3.104, -18.362, 72.856, -209.521, 3.966, -152.952]
  Set speed (1000.0 mm/s)
  MoveL 475 to (189, -575.99, 20) mm, rotated rx 180 ry 0 rz 90 deg; joints [-5.138, -18.208, 72.448, -225.975, 4.496, -138.111]
  Set speed (50.0 mm/s)
  MoveL 476 to (189, -575.99, 0) mm, rotated rx -180 ry 0 rz 90 deg; joints [-5.138, -17.345, 71.889, -223.33, 4.711, -140.764]
  MoveL 477 to (189, -575.99, 20) mm, rotated rx 180 ry 0 rz 90 deg; joints [-5.138, -18.208, 72.448, -225.975, 4.496, -138.111]
  Set speed (1000.0 mm/s)
  MoveL 478 to (189, -525.29, 20) mm, rotated rx -180 ry 0 rz 90 deg; joints [-5.264, -19.604, 76.191, -211.254, 6.39, -153]
  Set speed (50.0 mm/s)
  MoveL 479 to (189, -525.29, 0) mm, rotated rx -180 ry 0 rz 90 deg; joints [-5.264, -18.733, 75.641, -209.83, 6.666, -154.433]
  MoveL 480 to (189, -525.29, 20) mm, rotated rx -180 ry 0 rz 90 deg; joints [-5.264, -19.604, 76.191, -211.254, 6.39, -153]
  Set speed (1000.0 mm/s)
  MoveL 481 to (189, -474.6, 20) mm, rotated rx -180 ry 0 rz 90 deg; joints [-5.397, -20.893, 79.775, -203.715, 8.463, -160.714]
  Set speed (50.0 mm/s)
  MoveL 482 to (189, -474.6, 0) mm, rotated rx 180 ry 0 rz 90 deg; joints [-5.397, -20.012, 79.231, -202.836, 8.773, -161.603]
  MoveL 483 to (189, -474.6, 20) mm, rotated rx -180 ry 0 rz 90 deg; joints [-5.397, -20.893, 79.775, -203.715, 8.463, -160.714]
  Set speed (1000.0 mm/s)
  MoveL 484 to (189, -423.9, 20) mm, rotated rx -180 ry 0 rz 90 deg; joints [-5.536, -22.082, 83.22, -199.293, 10.589, -165.32]
  Set speed (50.0 mm/s)
  MoveL 485 to (189, -423.9, 0) mm, rotated rx -180 ry 0 rz 90 deg; joints [-5.536, -21.189, 82.68, -198.688, 10.923, -165.936]
  MoveL 486 to (189, -423.9, 20) mm, rotated rx -180 ry 0 rz 90 deg; joints [-5.536, -22.082, 83.22, -199.293, 10.589, -165.32]
  Set speed (1000.0 mm/s)
  MoveL 487 to (189, -373.21, 20) mm, rotated rx 180 ry 0 rz 90 deg; joints [-5.683, -23.178, 86.541, -196.43, 12.729, -168.375]
  Set speed (50.0 mm/s)
  MoveL 488 to (189, -373.21, 0) mm, rotated rx 180 ry 0 rz 90 deg; joints [-5.683, -22.271, 86.003, -195.981, 13.083, -168.836]
  MoveL 489 to (189, -373.21, 20) mm, rotated rx 180 ry 0 rz 90 deg; joints [-5.683, -23.178, 86.541, -196.43, 12.729, -168.375]
  Set speed (1000.0 mm/s)
  MoveL 490 to (189, -322.51, 20) mm, rotated rx 180 ry 0 rz 90 deg; joints [-5.838, -24.183, 89.751, -194.442, 14.872, -170.566]
  Set speed (50.0 mm/s)
  MoveL 491 to (189, -322.51, 0) mm, rotated rx -180 ry 0 rz 90 deg; joints [-5.838, -23.261, 89.213, -194.09, 15.244, -170.93]
  MoveL 492 to (189, -322.51, 20) mm, rotated rx 180 ry 0 rz 90 deg; joints [-5.838, -24.183, 89.751, -194.442, 14.872, -170.566]
  Set speed (1000.0 mm/s)
  MoveL 493 to (189, -271.82, 20) mm, rotated rx 180 ry 0 rz 90 deg; joints [-6.002, -25.1, 92.859, -192.994, 17.016, -172.228]
  Set speed (50.0 mm/s)
  MoveL 494 to (189, -271.82, 0) mm, rotated rx 180 ry 0 rz 90 deg; joints [-6.002, -24.161, 92.319, -192.707, 17.405, -172.528]
  MoveL 495 to (189, -271.82, 20) mm, rotated rx 180 ry 0 rz 90 deg; joints [-6.002, -25.1, 92.859, -192.994, 17.016, -172.228]
  Set speed (1000.0 mm/s)
  MoveL 496 to (189, -221.12, 20) mm, rotated rx 180 ry 0 rz 90 deg; joints [-6.174, -25.931, 95.874, -191.9, 19.163, -173.548]
  Set speed (50.0 mm/s)
  MoveL 497 to (189, -221.12, 0) mm, rotated rx -180 ry 0 rz 90 deg; joints [-6.174, -24.975, 95.331, -191.66, 19.568, -173.803]
  MoveL 498 to (189, -221.12, 20) mm, rotated rx 180 ry 0 rz 90 deg; joints [-6.174, -25.931, 95.874, -191.9, 19.163, -173.548]
  Set speed (1000.0 mm/s)
  MoveL 499 to (189, -170.43, 20) mm, rotated rx 180 ry 0 rz 90 deg; joints [-6.357, -26.675, 98.802, -191.052, 21.315, -174.636]
  Set speed (50.0 mm/s)
  MoveL 500 to (189, -170.43, 0) mm, rotated rx 180 ry 0 rz 90 deg; joints [-6.357, -25.7, 98.255, -190.846, 21.736, -174.857]
  MoveL 501 to (189, -170.43, 20) mm, rotated rx 180 ry 0 rz 90 deg; joints [-6.357, -26.675, 98.802, -191.052, 21.315, -174.636]
  Set speed (1000.0 mm/s)
  MoveL 502 to (189, -119.73, 20) mm, rotated rx 180 ry 0 rz 90 deg; joints [-6.552, -27.332, 101.65, -190.383, 23.479, -175.561]
  Set speed (50.0 mm/s)
  MoveL 503 to (189, -119.73, 0) mm, rotated rx -180 ry 0 rz 90 deg; joints [-6.552, -26.336, 101.097, -190.203, 23.914, -175.757]
  MoveL 504 to (189, -119.73, 20) mm, rotated rx 180 ry 0 rz 90 deg; joints [-6.552, -27.332, 101.65, -190.383, 23.479, -175.561]
  Set speed (1000.0 mm/s)
  MoveL 505 to (189, -69.03, 20) mm, rotated rx 180 ry 0 rz 90 deg; joints [-6.758, -27.9, 104.423, -189.848, 25.658, -176.369]
  Set speed (50.0 mm/s)
  MoveL 506 to (189, -69.03, 0) mm, rotated rx 180 ry 0 rz 90 deg; joints [-6.758, -26.883, 103.862, -189.688, 26.108, -176.546]
  MoveL 507 to (189, -69.03, 20) mm, rotated rx 180 ry 0 rz 90 deg; joints [-6.758, -27.9, 104.423, -189.848, 25.658, -176.369]
  Set speed (1000.0 mm/s)
  MoveL 508 to (189, -18.34, 20) mm, rotated rx -180 ry 0 rz 90 deg; joints [-6.978, -28.375, 107.122, -189.416, 27.858, -177.092]
  Set speed (50.0 mm/s)
  MoveL 509 to (189, -18.34, 0) mm, rotated rx -180 ry 0 rz 90 deg; joints [-6.978, -27.336, 106.553, -189.273, 28.323, -177.254]
  MoveL 510 to (189, -18.34, 20) mm, rotated rx -180 ry 0 rz 90 deg; joints [-6.978, -28.375, 107.122, -189.416, 27.858, -177.092]
  Set speed (1000.0 mm/s)
  MoveL 511 to (189, 32.36, 20) mm, rotated rx 180 ry 0 rz 90 deg; joints [-7.212, -28.755, 109.751, -189.068, 30.085, -177.754]
  Set speed (50.0 mm/s)
  MoveL 512 to (189, 32.36, 0) mm, rotated rx -180 ry 0 rz 90 deg; joints [-7.212, -27.692, 109.173, -188.938, 30.564, -177.904]
  MoveL 513 to (189, 32.36, 20) mm, rotated rx 180 ry 0 rz 90 deg; joints [-7.212, -28.755, 109.751, -189.068, 30.085, -177.754]
  Set speed (1000.0 mm/s)
  MoveL 514 to (189, 83.05, 20) mm, rotated rx 180 ry 0 rz 90 deg; joints [-7.463, -29.035, 112.313, -188.788, 32.345, -178.372]
  Set speed (50.0 mm/s)
  MoveL 515 to (189, 83.05, 0) mm, rotated rx -180 ry 0 rz 90 deg; joints [-7.463, -27.948, 111.724, -188.669, 32.837, -178.512]
  MoveL 516 to (189, 83.05, 20) mm, rotated rx 180 ry 0 rz 90 deg; joints [-7.463, -29.035, 112.313, -188.788, 32.345, -178.372]
  Set speed (1000.0 mm/s)
  MoveL 517 to (189, 133.75, 20) mm, rotated rx 180 ry 0 rz 90 deg; joints [-7.731, -29.21, 114.809, -188.565, 34.644, -178.96]
  Set speed (50.0 mm/s)
  MoveL 518 to (189, 133.75, 0) mm, rotated rx -180 ry 0 rz 90 deg; joints [-7.731, -28.097, 114.208, -188.456, 35.149, -179.092]
  MoveL 519 to (189, 133.75, 20) mm, rotated rx 180 ry 0 rz 90 deg; joints [-7.731, -29.21, 114.809, -188.565, 34.644, -178.96]
  Set speed (1000.0 mm/s)
  MoveL 520 to (189, 184.44, 20) mm, rotated rx -180 ry 0 rz 90 deg; joints [-8.019, -29.272, 117.239, -188.391, 36.988, -179.529]
  Set speed (50.0 mm/s)
  MoveL 521 to (189, 184.44, 0) mm, rotated rx 180 ry 0 rz 90 deg; joints [-8.019, -28.134, 116.624, -188.291, 37.506, -179.654]
  MoveL 522 to (189, 184.44, 20) mm, rotated rx -180 ry 0 rz 90 deg; joints [-8.019, -29.272, 117.239, -188.391, 36.988, -179.529]
  Set speed (1000.0 mm/s)
  MoveL 523 to (189, 235.14, 20) mm, rotated rx -180 ry 0 rz 90 deg; joints [-8.33, -29.215, 119.604, -188.261, 39.385, -180.089]
  Set speed (50.0 mm/s)
  MoveL 524 to (189, 235.14, 0) mm, rotated rx -180 ry 0 rz 90 deg; joints [-8.33, -28.05, 118.975, -188.169, 39.915, -180.209]
  MoveL 525 to (189, 235.14, 20) mm, rotated rx -180 ry 0 rz 90 deg; joints [-8.33, -29.215, 119.604, -188.261, 39.385, -180.089]
  Set speed (1000.0 mm/s)
  MoveL 526 to (189, 285.84, 20) mm, rotated rx 180 ry 0 rz 90 deg; joints [-8.666, -29.029, 121.903, -188.172, 41.843, -180.649]
  Set speed (50.0 mm/s)
  MoveL 527 to (189, 285.84, 0) mm, rotated rx -180 ry 0 rz 90 deg; joints [-8.666, -27.838, 121.257, -188.086, 42.383, -180.764]
  MoveL 528 to (189, 285.84, 20) mm, rotated rx 180 ry 0 rz 90 deg; joints [-8.666, -29.029, 121.903, -188.172, 41.843, -180.649]
  Set speed (1000.0 mm/s)
  MoveL 529 to (189, 336.53, 20) mm, rotated rx -180 ry 0 rz 90 deg; joints [-9.029, -28.705, 124.133, -188.119, 44.368, -181.217]
  Set speed (50.0 mm/s)
  MoveL 530 to (189, 336.53, 0) mm, rotated rx -180 ry 0 rz 90 deg; joints [-9.029, -27.488, 123.47, -188.041, 44.916, -181.327]
  MoveL 531 to (189, 336.53, 20) mm, rotated rx -180 ry 0 rz 90 deg; joints [-9.029, -28.705, 124.133, -188.119, 44.368, -181.217]
  Set speed (1000.0 mm/s)
  MoveL 532 to (189, 387.23, 20) mm, rotated rx 180 ry 0 rz 90 deg; joints [-9.424, -28.231, 126.294, -188.104, 46.97, -181.8]
  Set speed (50.0 mm/s)
  MoveL 533 to (189, 387.23, 0) mm, rotated rx -180 ry 0 rz 90 deg; joints [-9.424, -26.989, 125.612, -188.031, 47.525, -181.908]
  MoveL 534 to (189, 387.23, 20) mm, rotated rx 180 ry 0 rz 90 deg; joints [-9.424, -28.231, 126.294, -188.104, 46.97, -181.8]
  Set speed (1000.0 mm/s)
  MoveL 535 to (189, 437.92, 20) mm, rotated rx -180 ry 0 rz 90 deg; joints [-9.855, -27.596, 128.383, -188.124, 49.656, -182.409]
  Set speed (50.0 mm/s)
  MoveL 536 to (189, 437.92, 0) mm, rotated rx -180 ry 0 rz 90 deg; joints [-9.855, -26.329, 127.68, -188.057, 50.215, -182.512]
  MoveL 537 to (189, 437.92, 20) mm, rotated rx -180 ry 0 rz 90 deg; joints [-9.855, -27.596, 128.383, -188.124, 49.656, -182.409]
  Set speed (1000.0 mm/s)
  MoveL 538 to (189, 488.62, 20) mm, rotated rx 180 ry 0 rz 90 deg; joints [-10.326, -26.786, 130.395, -188.182, 52.436, -183.05]
  Set speed (50.0 mm/s)
  MoveL 539 to (189, 488.62, 0) mm, rotated rx -180 ry 0 rz 90 deg; joints [-10.326, -25.497, 129.671, -188.12, 52.996, -183.151]
  MoveL 540 to (189, 488.62, 20) mm, rotated rx 180 ry 0 rz 90 deg; joints [-10.326, -26.786, 130.395, -188.182, 52.436, -183.05]
  Set speed (1000.0 mm/s)
  MoveL 541 to (189, 539.31, 20) mm, rotated rx -180 ry 0 rz 90 deg; joints [-10.844, -25.787, 132.326, -188.279, 55.317, -183.734]
  Set speed (50.0 mm/s)
  MoveL 542 to (189, 539.31, 0) mm, rotated rx 180 ry 0 rz 90 deg; joints [-10.844, -24.477, 131.579, -188.223, 55.873, -183.832]
  MoveL 543 to (189, 539.31, 20) mm, rotated rx -180 ry 0 rz 90 deg; joints [-10.844, -25.787, 132.326, -188.279, 55.317, -183.734]
  Set speed (1000.0 mm/s)
  MoveL 544 to (189, 590.01, 20) mm, rotated rx 180 ry 0 rz 90 deg; joints [-11.417, -24.583, 134.171, -188.418, 58.308, -184.473]
  Set speed (50.0 mm/s)
  MoveL 545 to (189, 590.01, 0) mm, rotated rx 180 ry 0 rz 90 deg; joints [-11.417, -23.257, 133.4, -188.369, 58.856, -184.568]
  MoveL 546 to (189, 590.01, 20) mm, rotated rx 180 ry 0 rz 90 deg; joints [-11.417, -24.583, 134.171, -188.418, 58.308, -184.473]
  MoveL 547 to (189, 590.01, 20) mm, rotated rx 180 ry 0 rz 90 deg; joints [-11.417, -24.583, 134.171, -188.418, 58.308, -184.473]
  Set speed (1000.0 mm/s)
  MoveL 548 to (189, 590.01, 20) mm, rotated rx 180 ry 0 rz 90 deg; joints [-11.417, -24.583, 134.171, -188.418, 58.308, -184.473]
  MoveL 549 to (189, 590.01, 120) mm, rotated rx -180 ry 0 rz 90 deg; joints [-11.417, -31.583, 137.817, -188.748, 54.991, -183.874]
